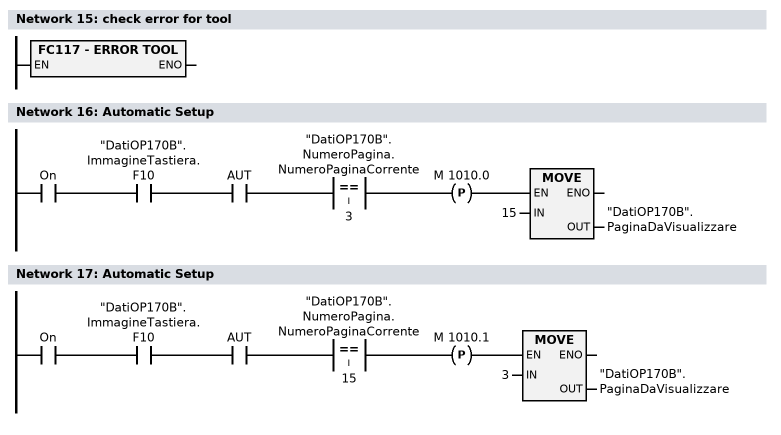
[picture p37: FC17 - OPERATOR PANNEL networks 15-17]
NETWORK
TITLE = check error for tool
      CALL  "FC117 - ERROR TOOL";
      NOP   0;
NETWORK
TITLE = Automatic Setup
      A     "On";
      A     "DatiOP170B".ImmagineTastiera.F10;
      A     "AUT";
      A(;
      L     "DatiOP170B".NumeroPagina.NumeroPaginaCorrente;
      L     3;
      ==I;
      );
      FP    M 1010.0;
      JNB   _00d;
      L     15;
      T     "DatiOP170B".PaginaDaVisualizzare;
_00d: NOP   0;
NETWORK
TITLE = Automatic Setup
      A     "On";
      A     "DatiOP170B".ImmagineTastiera.F10;
      A     "AUT";
      A(;
      L     "DatiOP170B".NumeroPagina.NumeroPaginaCorrente;
      L     15;
      ==I;
      );
      FP    M 1010.1;
      JNB   _00e;
      L     3;
      T     "DatiOP170B".PaginaDaVisualizzare;
_00e: NOP   0;
END_FUNCTION

FUNCTION "FC18 - OUTPUTS" : VOID	// FC 18
TITLE = Outputs management
VERSION : 0.1
BEGIN
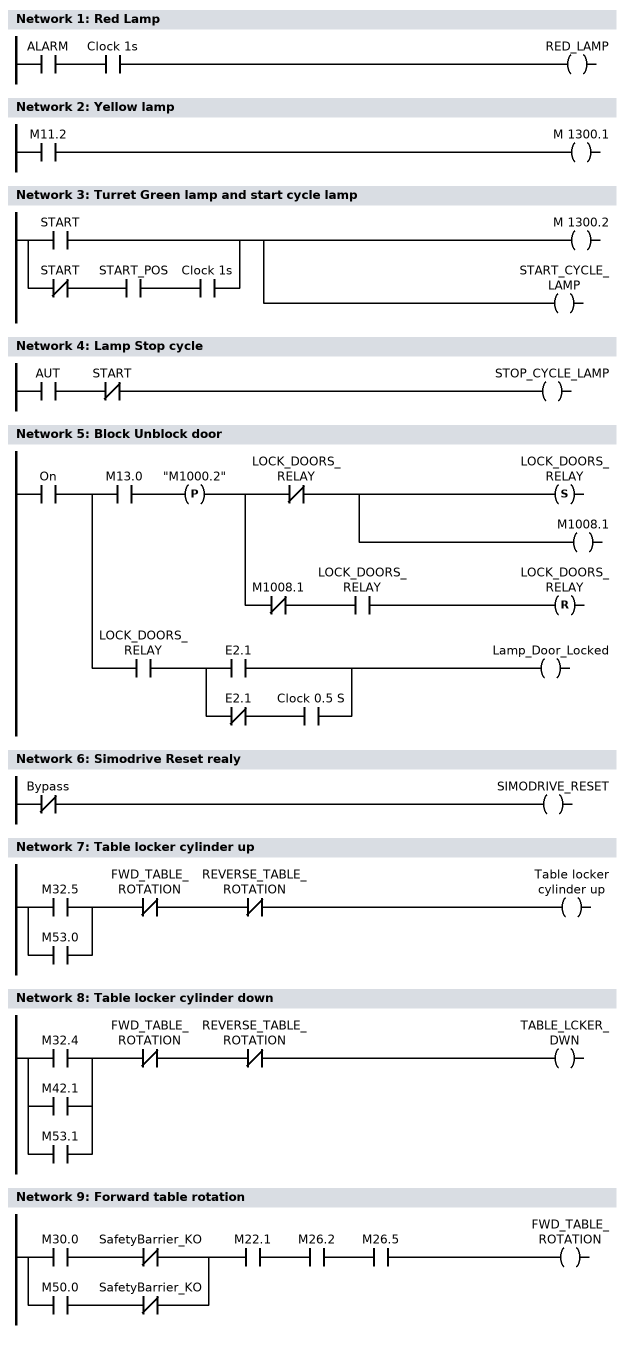
NETWORK
TITLE = Red Lamp
      A     "ALARM";
      A     "Clock 1s";
      =     "RED_LAMP";
NETWORK
TITLE = Yellow lamp
      A     "M11.2";
      =     M 1300.1;
NETWORK
TITLE = Turret Green lamp and start cycle lamp
      O     "START";
      O;
      AN    "START";
      A     "START_POS";
      A     "Clock 1s";
      =     M 1300.2;
      =     "START_CYCLE_LAMP";
NETWORK
TITLE = Lamp Stop cycle
      A     "AUT";
      AN    "START";
      =     "STOP_CYCLE_LAMP";
NETWORK
TITLE = Block Unblock door
//light ON = door lock
      A     "On";
      =     L 0.0;
      A     L 0.0;
      A     "M13.0";
      FP    "M1000.2";
      =     L 0.1;
      A     L 0.1;
      AN    "LOCK_DOORS_RELAY";
      S     "LOCK_DOORS_RELAY";
      =     "M1008.1";
      A     L 0.1;
      AN    "M1008.1";
      A     "LOCK_DOORS_RELAY";
      R     "LOCK_DOORS_RELAY";
      A     L 0.0;
      A     "LOCK_DOORS_RELAY";
      A(;
      O     "E2.1";
      O;
      AN    "E2.1";
      A     "Clock 0.5 S";
      );
      =     "Lamp_Door_Locked";
NETWORK
TITLE = Simodrive Reset realy
      AN    "Bypass";
      =     "SIMODRIVE_RESET";
NETWORK
TITLE = Table locker cylinder up
      A(;
      O     "M32.5";
      O     "M53.0";
      );
      AN    "FWD_TABLE_ROTATION";
      AN    "REVERSE_TABLE_ROTATION";
      =     "Table locker cylinder up";
NETWORK
TITLE = Table locker cylinder down
      A(;
      O     "M32.4";
      O     "M42.1";
      O     "M53.1";
      );
      AN    "FWD_TABLE_ROTATION";
      AN    "REVERSE_TABLE_ROTATION";
      =     "TABLE_LCKER_DWN";
NETWORK
TITLE = Forward table rotation
      A(;
      A     "M30.0";
      AN    "SafetyBarrier_KO";
      O;
      A     "M50.0";
      AN    "SafetyBarrier_KO";
      );
      A     "M22.1";
      A     "M26.2";
      A     "M26.5";
      =     "FWD_TABLE_ROTATION";
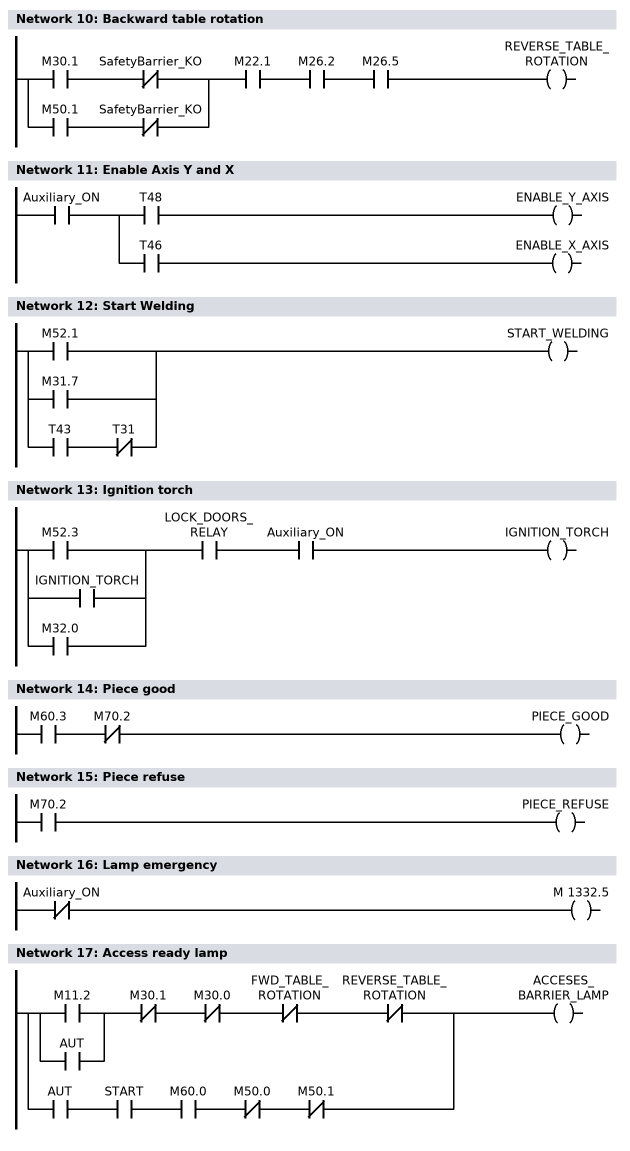
NETWORK
TITLE = Backward table rotation
      A(;
      A     "M30.1";
      AN    "SafetyBarrier_KO";
      O;
      A     "M50.1";
      AN    "SafetyBarrier_KO";
      );
      A     "M22.1";
      A     "M26.2";
      A     "M26.5";
      =     "REVERSE_TABLE_ROTATION";
NETWORK
TITLE = Enable Axis Y and X
      A     "Auxiliary_ON";
      =     L 0.0;
      A     L 0.0;
      A     "T48";
      =     "ENABLE_Y_AXIS";
      A     L 0.0;
      A     "T46";
      =     "ENABLE_X_AXIS";
NETWORK
TITLE = Start Welding
      O     "M52.1";
      O     "M31.7";
      O;
      A     "T43";
      AN    "T31";
      =     "START_WELDING";
NETWORK
TITLE = Ignition torch
      A(;
      O     "M52.3";
      O     "IGNITION_TORCH";
      O     "M32.0";
      );
      A     "LOCK_DOORS_RELAY";
      A     "Auxiliary_ON";
      =     "IGNITION_TORCH";
NETWORK
TITLE = Piece good
      A     "M60.3";
      AN    "M70.2";
      =     "PIECE_GOOD";
NETWORK
TITLE = Piece refuse
      A     "M70.2";
      =     "PIECE_REFUSE";
NETWORK
TITLE = Lamp emergency
      AN    "Auxiliary_ON";
      =     M 1332.5;
NETWORK
TITLE = Access ready lamp
      A(;
      O     "M11.2";
      O     "AUT";
      );
      AN    "M30.1";
      AN    "M30.0";
      AN    "FWD_TABLE_ROTATION";
      AN    "REVERSE_TABLE_ROTATION";
      O;
      A     "AUT";
      A     "START";
      A     "M60.0";
      AN    "M50.0";
      AN    "M50.1";
      =     "ACCESES_BARRIER_LAMP";
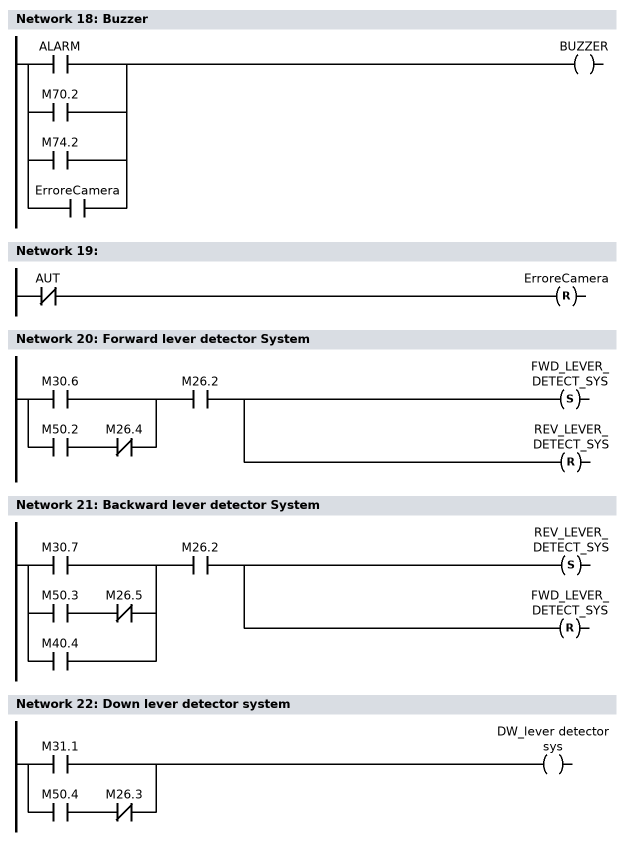
NETWORK
TITLE = Buzzer
//"Off"
      O     "ALARM";
      O     "M70.2";
      O     "M74.2";
      O     "ErroreCamera";
      =     "BUZZER";
NETWORK
TITLE =
      AN    "AUT";
      R     "ErroreCamera";
NETWORK
TITLE = Forward lever detector System
      A(;
      O     "M30.6";
      O;
      A     "M50.2";
      AN    "M26.4";
      );
      A     "M26.2";
      S     "FWD_LEVER_DETECT_SYS";
      R     "REV_LEVER_DETECT_SYS";
NETWORK
TITLE = Backward lever detector System
      A(;
      O     "M30.7";
      O;
      A     "M50.3";
      AN    "M26.5";
      O     "M40.4";
      );
      A     "M26.2";
      S     "REV_LEVER_DETECT_SYS";
      R     "FWD_LEVER_DETECT_SYS";
NETWORK
TITLE = Down lever detector system
      O     "M31.1";
      O;
      A     "M50.4";
      AN    "M26.3";
      =     "DW_lever detector sys";
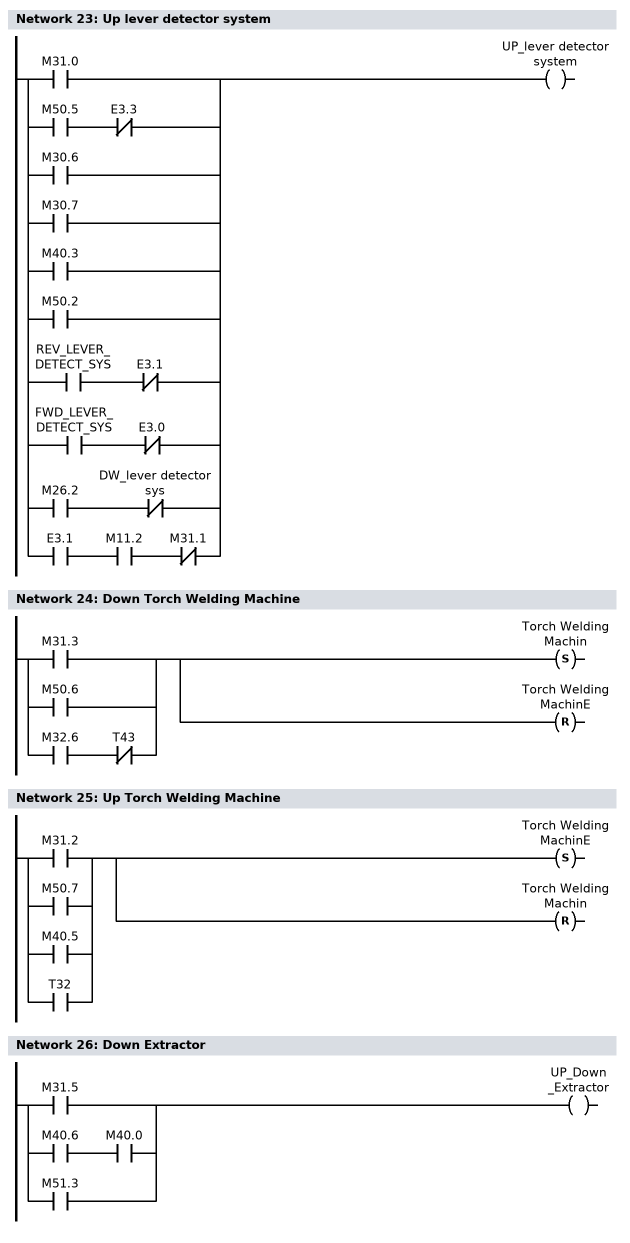
NETWORK
TITLE = Up lever detector system
      O     "M31.0";
      O;
      A     "M50.5";
      AN    "E3.3";
      O     "M30.6";
      O     "M30.7";
      O     "M40.3";
      O     "M50.2";
      O;
      A     "REV_LEVER_DETECT_SYS";
      AN    "E3.1";
      O;
      A     "FWD_LEVER_DETECT_SYS";
      AN    "E3.0";
      O;
      A     "M26.2";
      AN    "DW_lever detector sys";
      O;
      A     "E3.1";
      A     "M11.2";
      AN    "M31.1";
      =     "UP_lever detector system";
NETWORK
TITLE = Down Torch Welding Machine
      O     "M31.3";
      O     "M50.6";
      O;
      A     "M32.6";
      AN    "T43";
      S     "Torch Welding Machin";
      R     "Torch Welding MachinE";
NETWORK
TITLE = Up Torch Welding Machine
      O     "M31.2";
      O     "M50.7";
      O     "M40.5";
      O     "T32";
      S     "Torch Welding MachinE";
      R     "Torch Welding Machin";
NETWORK
TITLE = Down Extractor
      O     "M31.5";
      O;
      A     "M40.6";
      A     "M40.0";
      O     "M51.3";
      =     "UP_Down _Extractor";
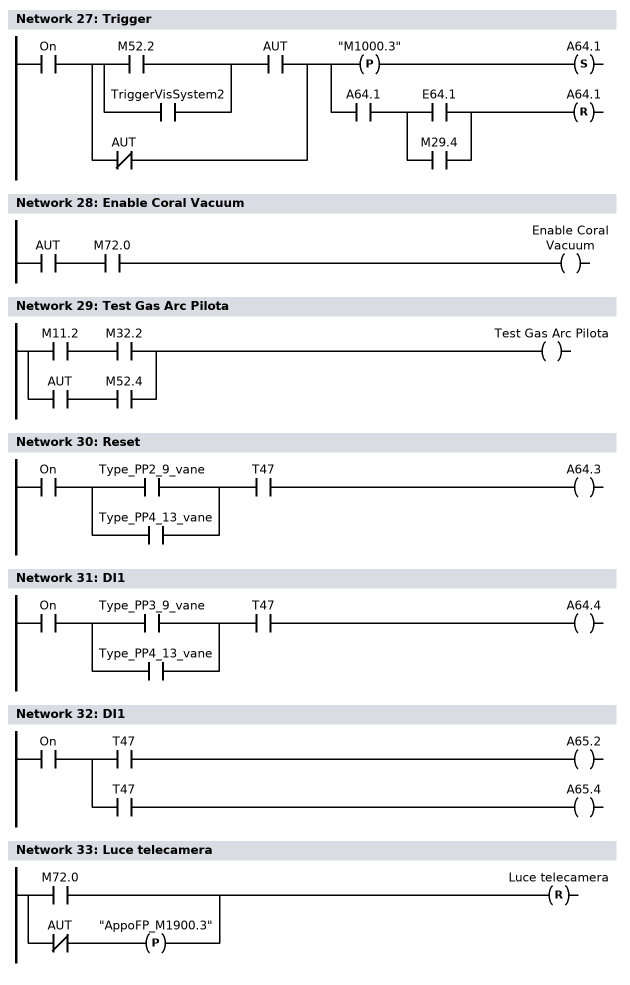
NETWORK
TITLE = Trigger
      A     "On";
      A(;
      A(;
      O     "M52.2";
      O     "TriggerVisSystem2";
      );
      A     "AUT";
      ON    "AUT";
      );
      =     L 0.0;
      A     L 0.0;
      FP    "M1000.3";
      S     "A64.1";
      A     L 0.0;
      A     "A64.1";
      A(;
      O     "E64.1";
      O     "M29.4";
      );
      R     "A64.1";
NETWORK
TITLE = Enable Coral Vacuum
      A     "AUT";
      A     "M72.0";
      =     "Enable Coral Vacuum";
NETWORK
TITLE = Test Gas Arc Pilota
//Test Arco Gas
      A     "M11.2";
      A     "M32.2";
      O;
      A     "AUT";
      A     "M52.4";
      =     "Test Gas Arc Pilota";
NETWORK
TITLE = Reset
//bit DI0 Select Scene TeleCam
      A     "On";
      A(;
      O     "Type_PP2_9_vane";
      O     "Type_PP4_13_vane";
      );
      A     "T47";
      =     "A64.3";
NETWORK
TITLE = DI1
//bit DI1 Select Scene TeleCam
      A     "On";
      A(;
      O     "Type_PP3_9_vane";
      O     "Type_PP4_13_vane";
      );
      A     "T47";
      =     "A64.4";
NETWORK
TITLE = DI1
//Select Scene Cam
      A     "On";
      =     L 0.0;
      A     L 0.0;
      A     "T47";
      =     "A65.2";
      A     L 0.0;
      A     "T47";
      =     "A65.4";
NETWORK
TITLE = Luce telecamera
      O     "M72.0";
      O(;
      AN    "AUT";
      FP    "AppoFP_M1900.3";
      );
      R     "Luce telecamera";
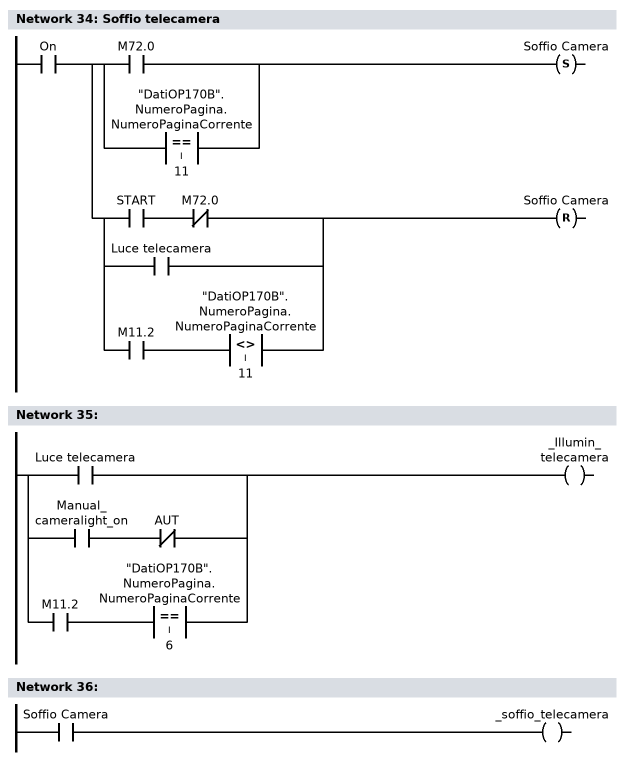
NETWORK
TITLE = Soffio telecamera
      A     "On";
      =     L 0.0;
      A     L 0.0;
      A(;
      O     "M72.0";
      O(;
      L     "DatiOP170B".NumeroPagina.NumeroPaginaCorrente;
      L     11;
      ==I;
      );
      );
      S     "Soffio Camera";
      A     L 0.0;
      A(;
      A     "START";
      AN    "M72.0";
      O     "Luce telecamera";
      O;
      A     "M11.2";
      A(;
      L     "DatiOP170B".NumeroPagina.NumeroPaginaCorrente;
      L     11;
      <>I;
      );
      );
      R     "Soffio Camera";
NETWORK
TITLE =
      O     "Luce telecamera";
      O;
      A     "Manual_cameralight_on";
      AN    "AUT";
      O;
      A     "M11.2";
      A(;
      L     "DatiOP170B".NumeroPagina.NumeroPaginaCorrente;
      L     6;
      ==I;
      );
      =     "_Illumin_telecamera";
NETWORK
TITLE =
      A     "Soffio Camera";
      =     "_soffio_telecamera";
END_FUNCTION

FUNCTION "FC19 - REPOSITIONING" : VOID	// FC 19
TITLE = Repositioning management
VERSION : 0.1
BEGIN
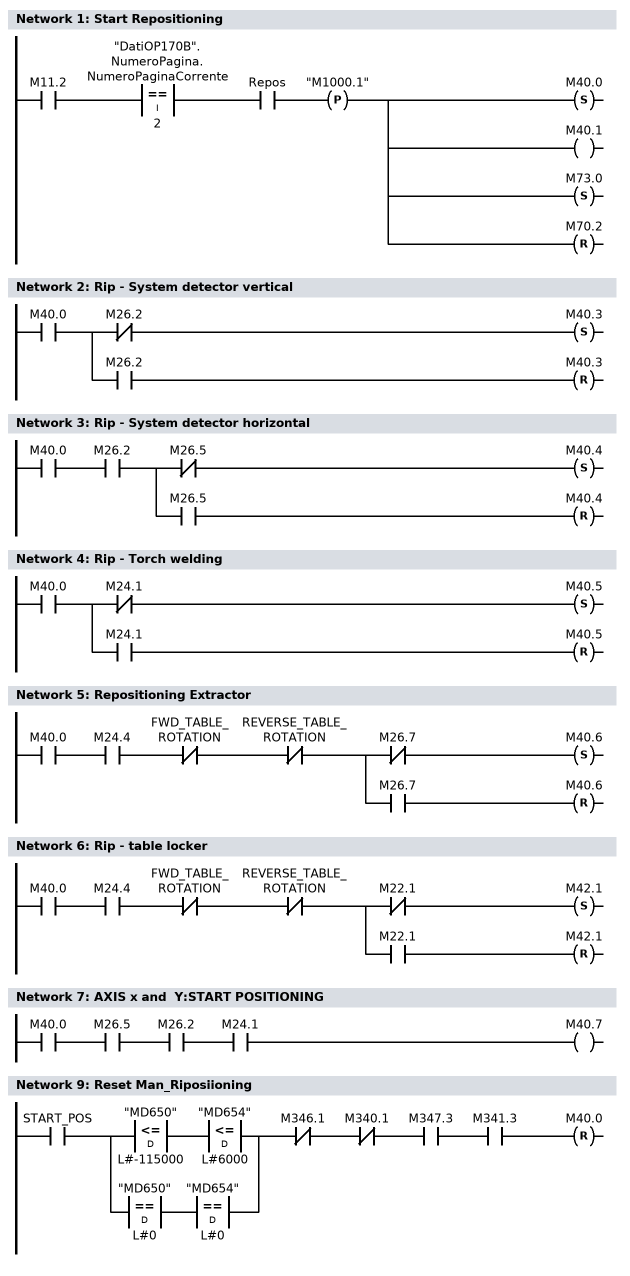
NETWORK
TITLE = Start Repositioning
      A     "M11.2";
      A(;
      L     "DatiOP170B".NumeroPagina.NumeroPaginaCorrente;
      L     2;
      ==I;
      );
      A     "Repos";
      FP    "M1000.1";
      S     "M40.0";
      =     "M40.1";
      S     "M73.0";
      R     "M70.2";
NETWORK
TITLE = Rip - System detector vertical
//ripositioning Table
      A     "M40.0";
      =     L 0.0;
      A     L 0.0;
      AN    "M26.2";
      S     "M40.3";
      A     L 0.0;
      A     "M26.2";
      R     "M40.3";
NETWORK
TITLE = Rip - System detector horizontal
//ripositioning Table
      A     "M40.0";
      A     "M26.2";
      =     L 0.0;
      A     L 0.0;
      AN    "M26.5";
      S     "M40.4";
      A     L 0.0;
      A     "M26.5";
      R     "M40.4";
NETWORK
TITLE = Rip - Torch welding
//ripositioning Table
      A     "M40.0";
      =     L 0.0;
      A     L 0.0;
      AN    "M24.1";
      S     "M40.5";
      A     L 0.0;
      A     "M24.1";
      R     "M40.5";
NETWORK
TITLE = Repositioning Extractor
      A     "M40.0";
      A     "M24.4";
      AN    "FWD_TABLE_ROTATION";
      AN    "REVERSE_TABLE_ROTATION";
      =     L 0.0;
      A     L 0.0;
      AN    "M26.7";
      S     "M40.6";
      A     L 0.0;
      A     "M26.7";
      R     "M40.6";
NETWORK
TITLE = Rip - table locker
      A     "M40.0";
      A     "M24.4";
      AN    "FWD_TABLE_ROTATION";
      AN    "REVERSE_TABLE_ROTATION";
      =     L 0.0;
      A     L 0.0;
      AN    "M22.1";
      S     "M42.1";
      A     L 0.0;
      A     "M22.1";
      R     "M42.1";
NETWORK
TITLE = AXIS x and  Y:START POSITIONING
      A     "M40.0";
      A     "M26.5";
      A     "M26.2";
      A     "M24.1";
      =     "M40.7";
NETWORK
TITLE = Reset Man_Riposiioning
//      U     "START_POS"
//      U(    
//      U(    
//      L     "MD650"
//      L     L#-115000
//      <=D   
//      )     
//      U(    
//      L     "MD654"
//      L     L#6000
//      <=D   
//      )     
//      O     
//      U(    
//      L     "MD650"
//      L     L#0
//      ==I   
//      )     
//      U(    
//      L     "MD654"
//      L     L#0
//      ==I   
//      )     
//      )     
//      UN    "M346.1"
//      UN    "M340.1"
//      U     "M347.3"
//      U     "M341.3"
//      R     "M40.0"
NETWORK
TITLE = Reset Man_Riposiioning
      A     "START_POS";
      A(;
      A(;
      L     "MD650";
      L     L#-115000;
      <=D;
      );
      A(;
      L     "MD654";
      L     L#6000;
      <=D;
      );
      O;
      A(;
      L     "MD650";
      L     L#0;
      ==D;
      );
      A(;
      L     "MD654";
      L     L#0;
      ==D;
      );
      );
      AN    "M346.1";
      AN    "M340.1";
      A     "M347.3";
      A     "M341.3";
      R     "M40.0";
NETWORK
TITLE =
END_FUNCTION

FUNCTION "FC50 - TEACH-IN" : VOID	// FC 50
TITLE = TEACH_IN
VERSION : 0.1
BEGIN
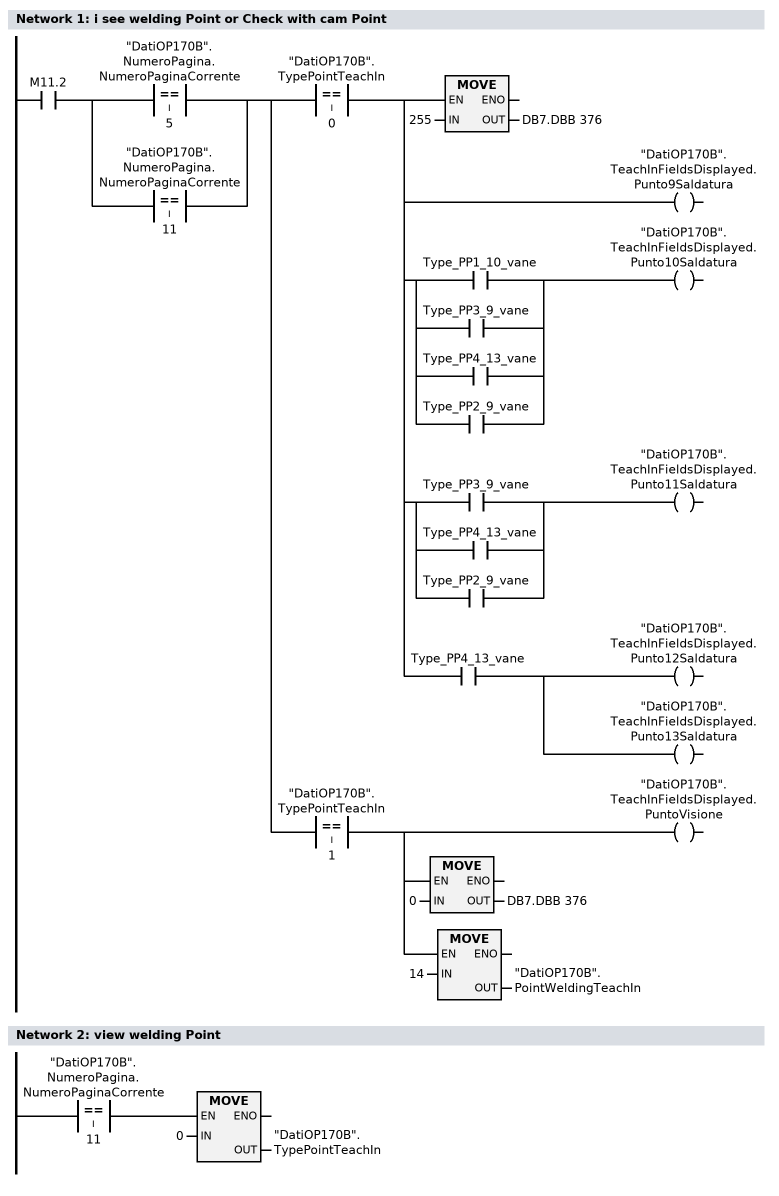
NETWORK
TITLE = i see welding Point or Check with cam Point
      A     "M11.2";
      A(;
      O(;
      L     "DatiOP170B".NumeroPagina.NumeroPaginaCorrente;
      L     5;
      ==I;
      );
      O(;
      L     "DatiOP170B".NumeroPagina.NumeroPaginaCorrente;
      L     11;
      ==I;
      );
      );
      =     L 0.0;
      A     L 0.0;
      A(;
      L     "DatiOP170B".TypePointTeachIn;
      L     0;
      ==I;
      );
      =     L 0.1;
      A     L 0.1;
      JNB   _001;
      L     255;
      T     DB7.DBB 376;
_001: NOP   0;
      A     L 0.1;
      BLD   102;
      =     "DatiOP170B".TeachInFieldsDisplayed.Punto9Saldatura;
      A     L 0.1;
      A(;
      O     "Type_PP1_10_vane";
      O     "Type_PP3_9_vane";
      O     "Type_PP4_13_vane";
      O     "Type_PP2_9_vane";
      );
      =     "DatiOP170B".TeachInFieldsDisplayed.Punto10Saldatura;
      A     L 0.1;
      A(;
      O     "Type_PP3_9_vane";
      O     "Type_PP4_13_vane";
      O     "Type_PP2_9_vane";
      );
      =     "DatiOP170B".TeachInFieldsDisplayed.Punto11Saldatura;
      A     L 0.1;
      A     "Type_PP4_13_vane";
      =     "DatiOP170B".TeachInFieldsDisplayed.Punto12Saldatura;
      =     "DatiOP170B".TeachInFieldsDisplayed.Punto13Saldatura;
      A     L 0.0;
      A(;
      L     "DatiOP170B".TypePointTeachIn;
      L     1;
      ==I;
      );
      =     L 0.1;
      A     L 0.1;
      BLD   102;
      =     "DatiOP170B".TeachInFieldsDisplayed.PuntoVisione;
      A     L 0.1;
      JNB   _002;
      L     0;
      T     DB7.DBB 376;
_002: NOP   0;
      A     L 0.1;
      JNB   _003;
      L     14;
      T     "DatiOP170B".PointWeldingTeachIn;
_003: NOP   0;
NETWORK
TITLE = view welding Point
      A(;
      L     "DatiOP170B".NumeroPagina.NumeroPaginaCorrente;
      L     11;
      ==I;
      );
      JNB   _004;
      L     0;
      T     "DatiOP170B".TypePointTeachIn;
_004: NOP   0;
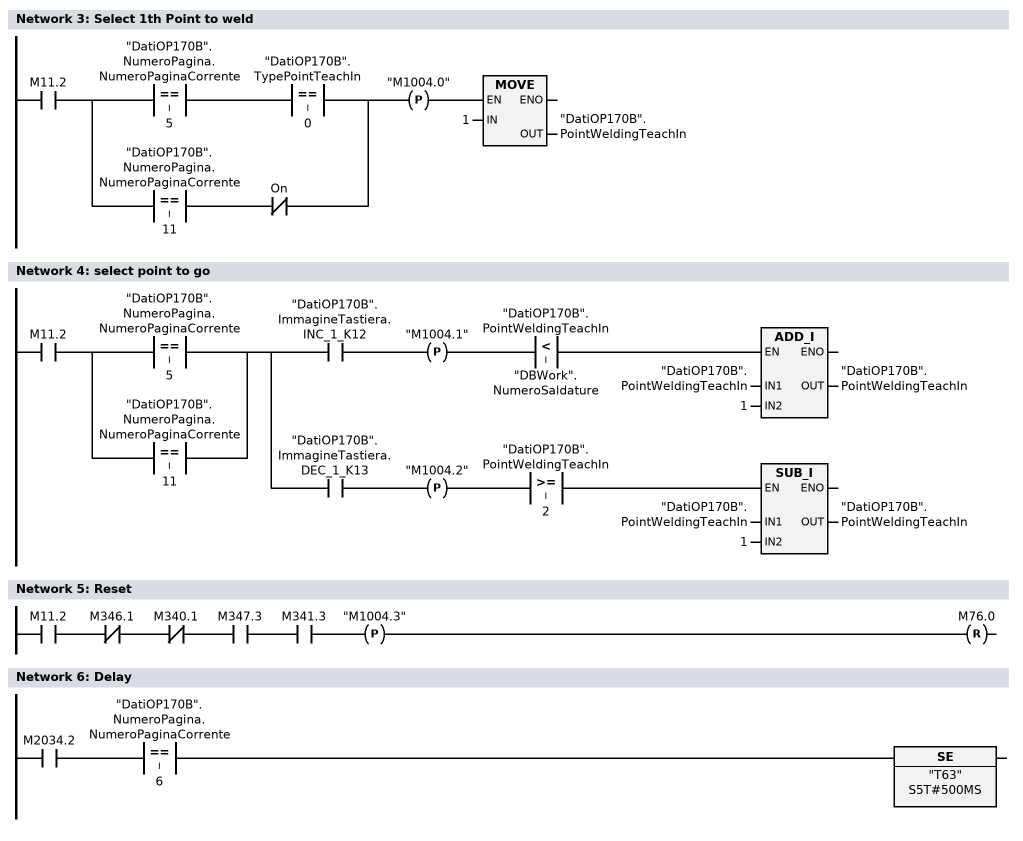
NETWORK
TITLE = Select 1th Point to weld
      A     "M11.2";
      A(;
      A(;
      L     "DatiOP170B".NumeroPagina.NumeroPaginaCorrente;
      L     5;
      ==I;
      );
      A(;
      L     "DatiOP170B".TypePointTeachIn;
      L     0;
      ==I;
      );
      O;
      A(;
      L     "DatiOP170B".NumeroPagina.NumeroPaginaCorrente;
      L     11;
      ==I;
      );
      AN    "On";
      );
      FP    "M1004.0";
      JNB   _005;
      L     1;
      T     "DatiOP170B".PointWeldingTeachIn;
_005: NOP   0;
NETWORK
TITLE = select point to go
      A     "M11.2";
      A(;
      O(;
      L     "DatiOP170B".NumeroPagina.NumeroPaginaCorrente;
      L     5;
      ==I;
      );
      O(;
      L     "DatiOP170B".NumeroPagina.NumeroPaginaCorrente;
      L     11;
      ==I;
      );
      );
      =     L 0.0;
      A     L 0.0;
      A     "DatiOP170B".ImmagineTastiera.INC_1_K12;
      FP    "M1004.1";
      A(;
      L     "DatiOP170B".PointWeldingTeachIn;
      L     "DBWork".NumeroSaldature;
      <I;
      );
      JNB   _006;
      L     "DatiOP170B".PointWeldingTeachIn;
      L     1;
      +I;
      T     "DatiOP170B".PointWeldingTeachIn;
_006: NOP   0;
      A     L 0.0;
      A     "DatiOP170B".ImmagineTastiera.DEC_1_K13;
      FP    "M1004.2";
      A(;
      L     "DatiOP170B".PointWeldingTeachIn;
      L     2;
      >=I;
      );
      JNB   _007;
      L     "DatiOP170B".PointWeldingTeachIn;
      L     1;
      -I;
      T     "DatiOP170B".PointWeldingTeachIn;
_007: NOP   0;
NETWORK
TITLE = Reset
      A     "M11.2";
      AN    "M346.1";
      AN    "M340.1";
      A     "M347.3";
      A     "M341.3";
      FP    "M1004.3";
      R     "M76.0";
NETWORK
TITLE = Delay
      A     "M2034.2";
      A(;
      L     "DatiOP170B".NumeroPagina.NumeroPaginaCorrente;
      L     6;
      ==I;
      );
      L     S5T#500MS;
      SE    "T63";
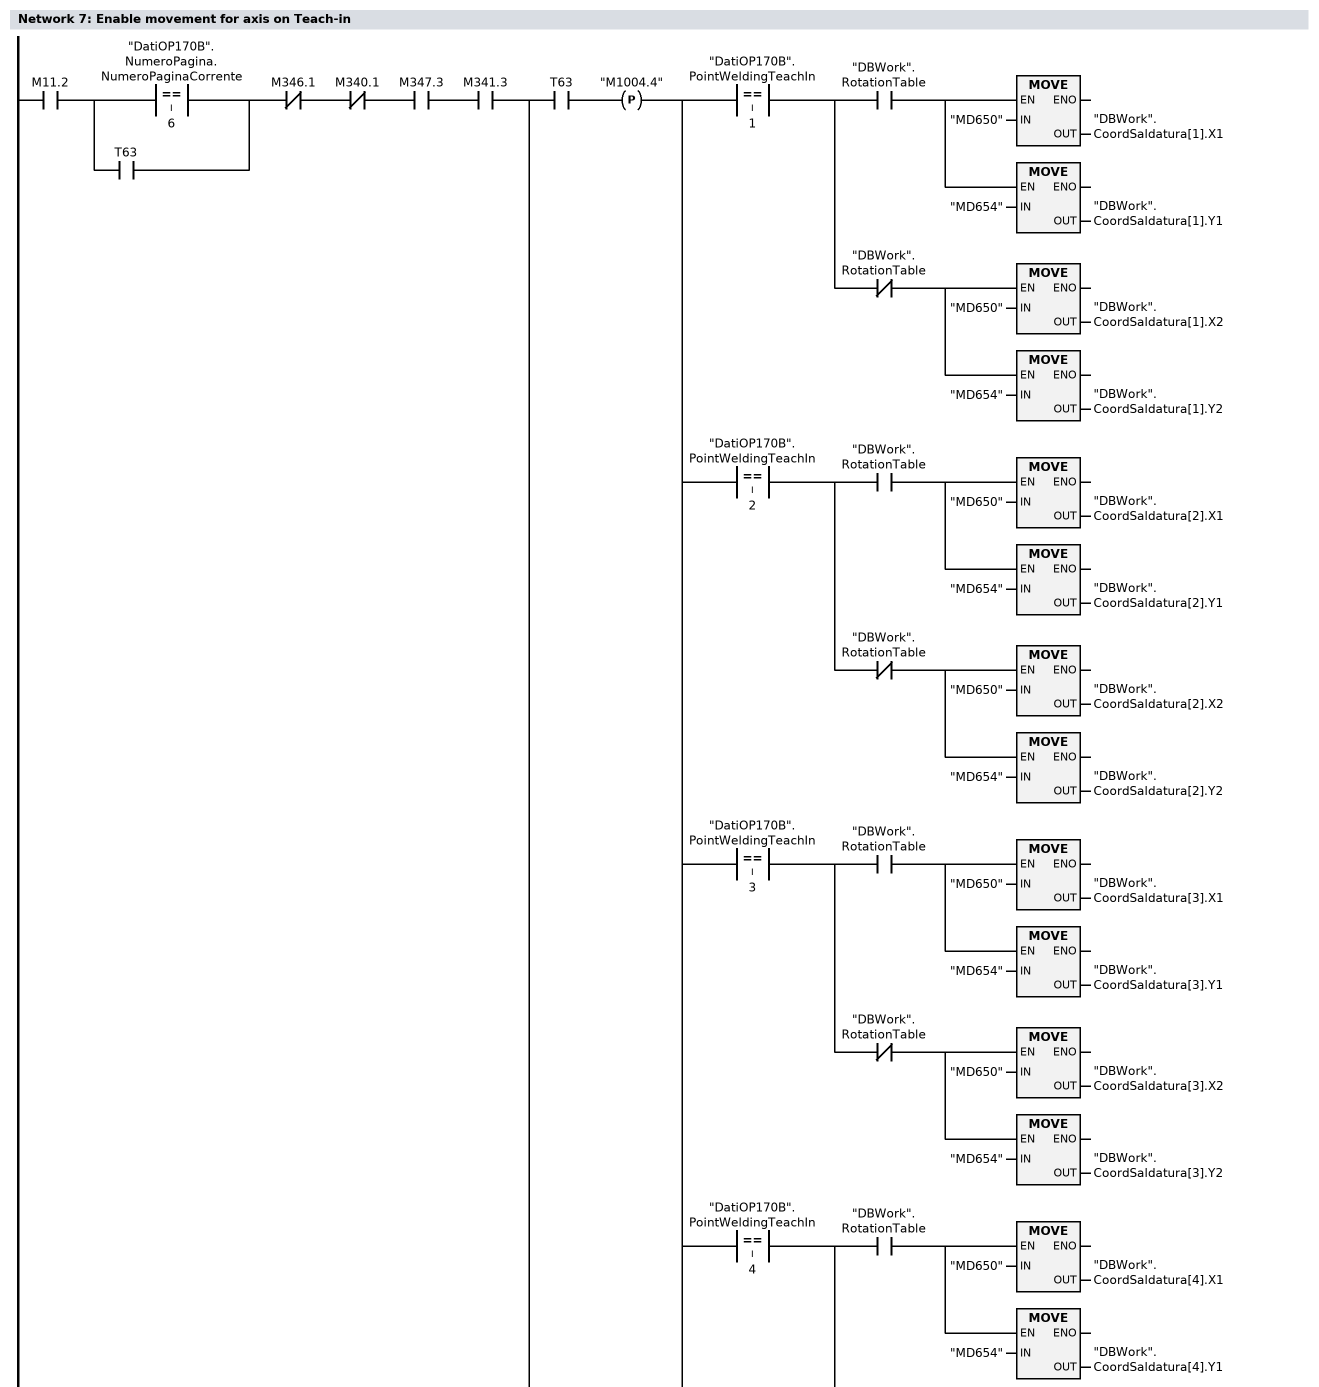
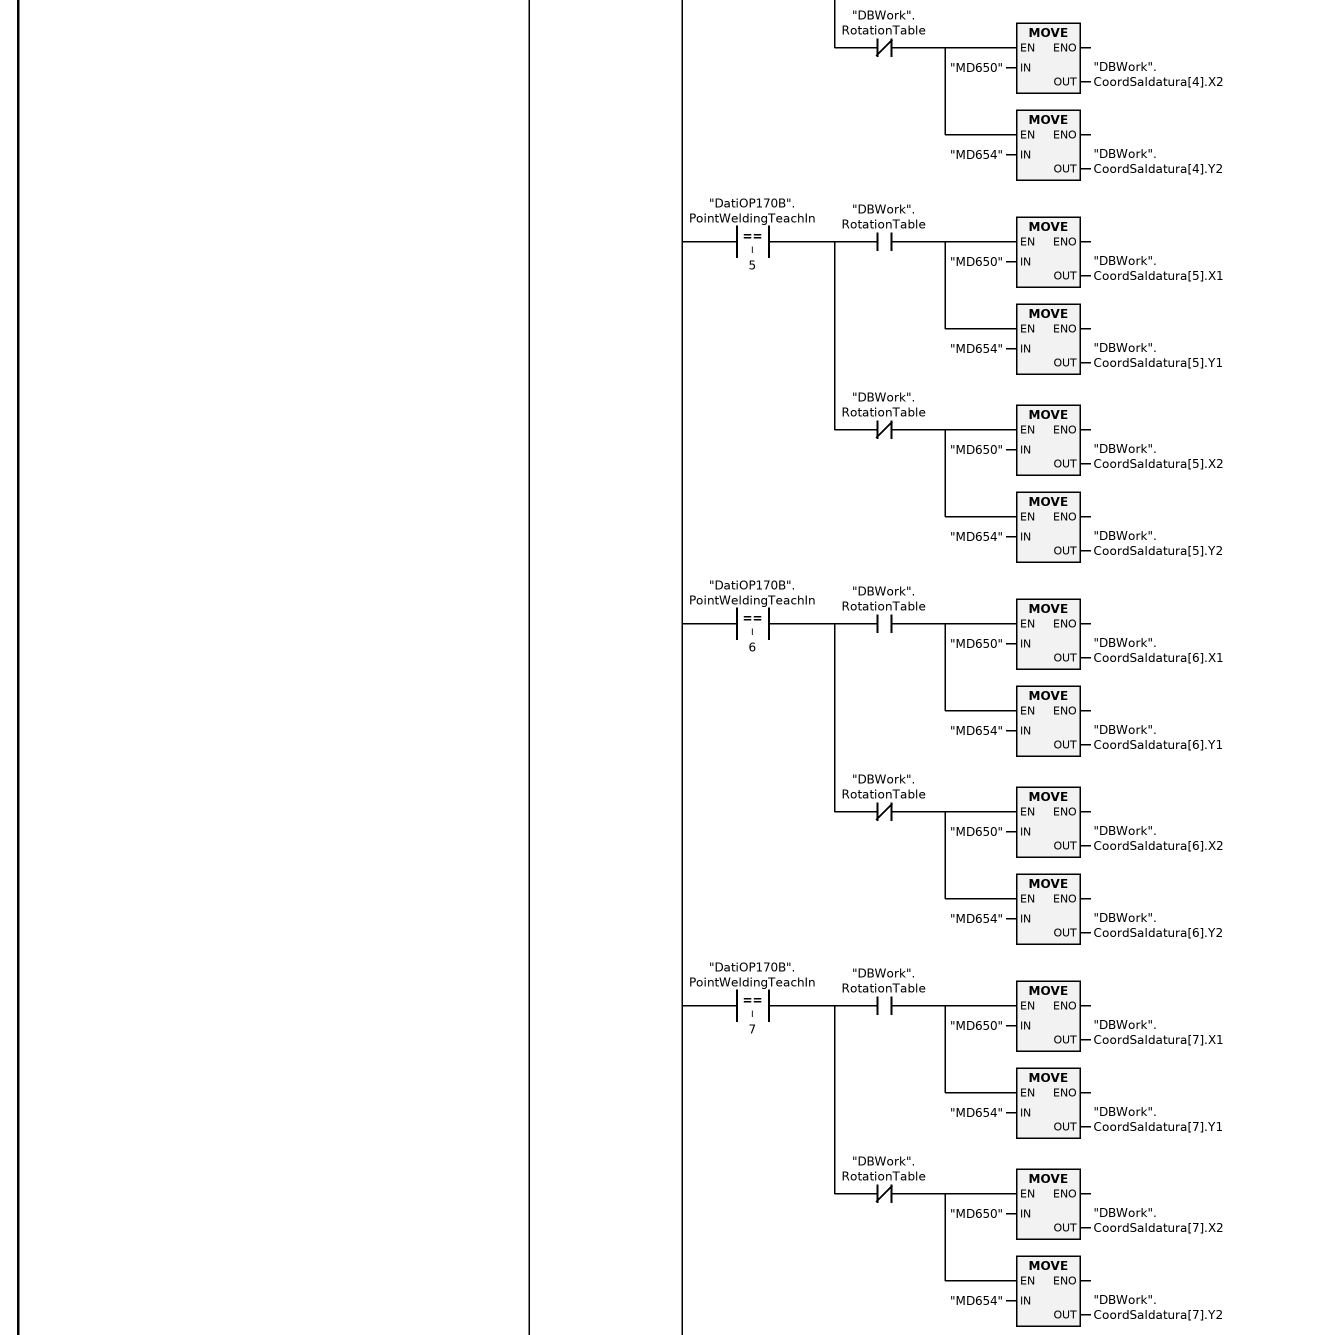
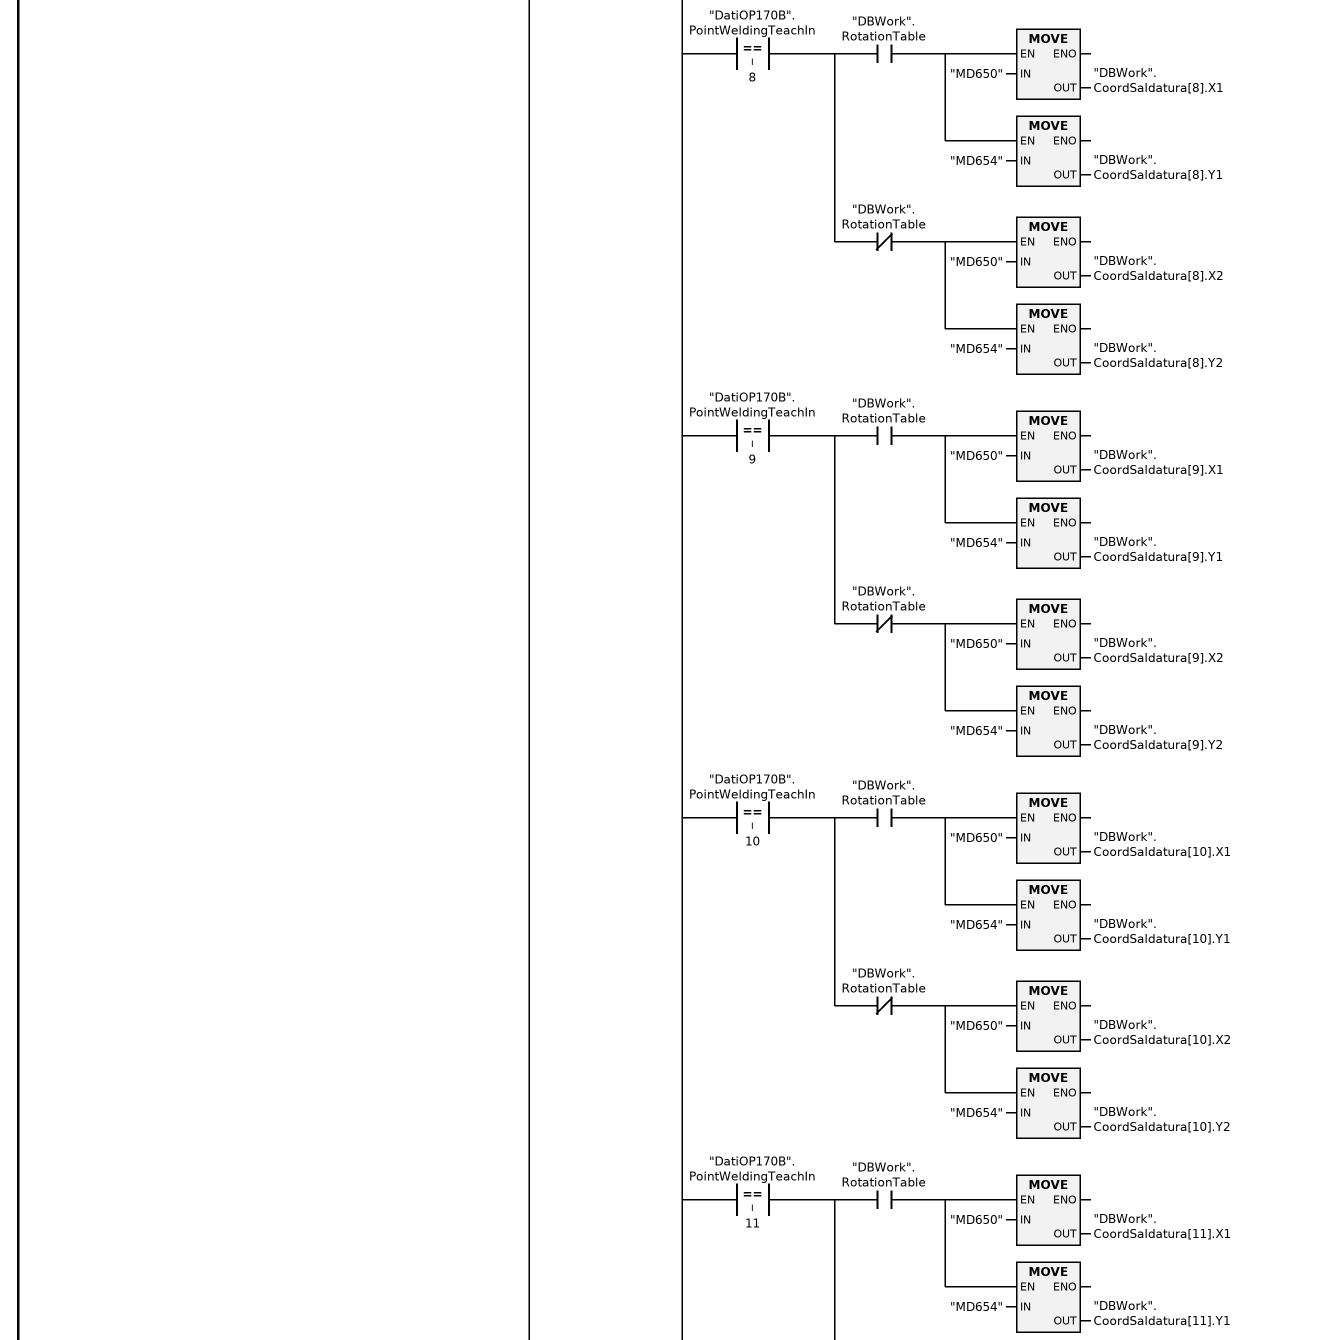
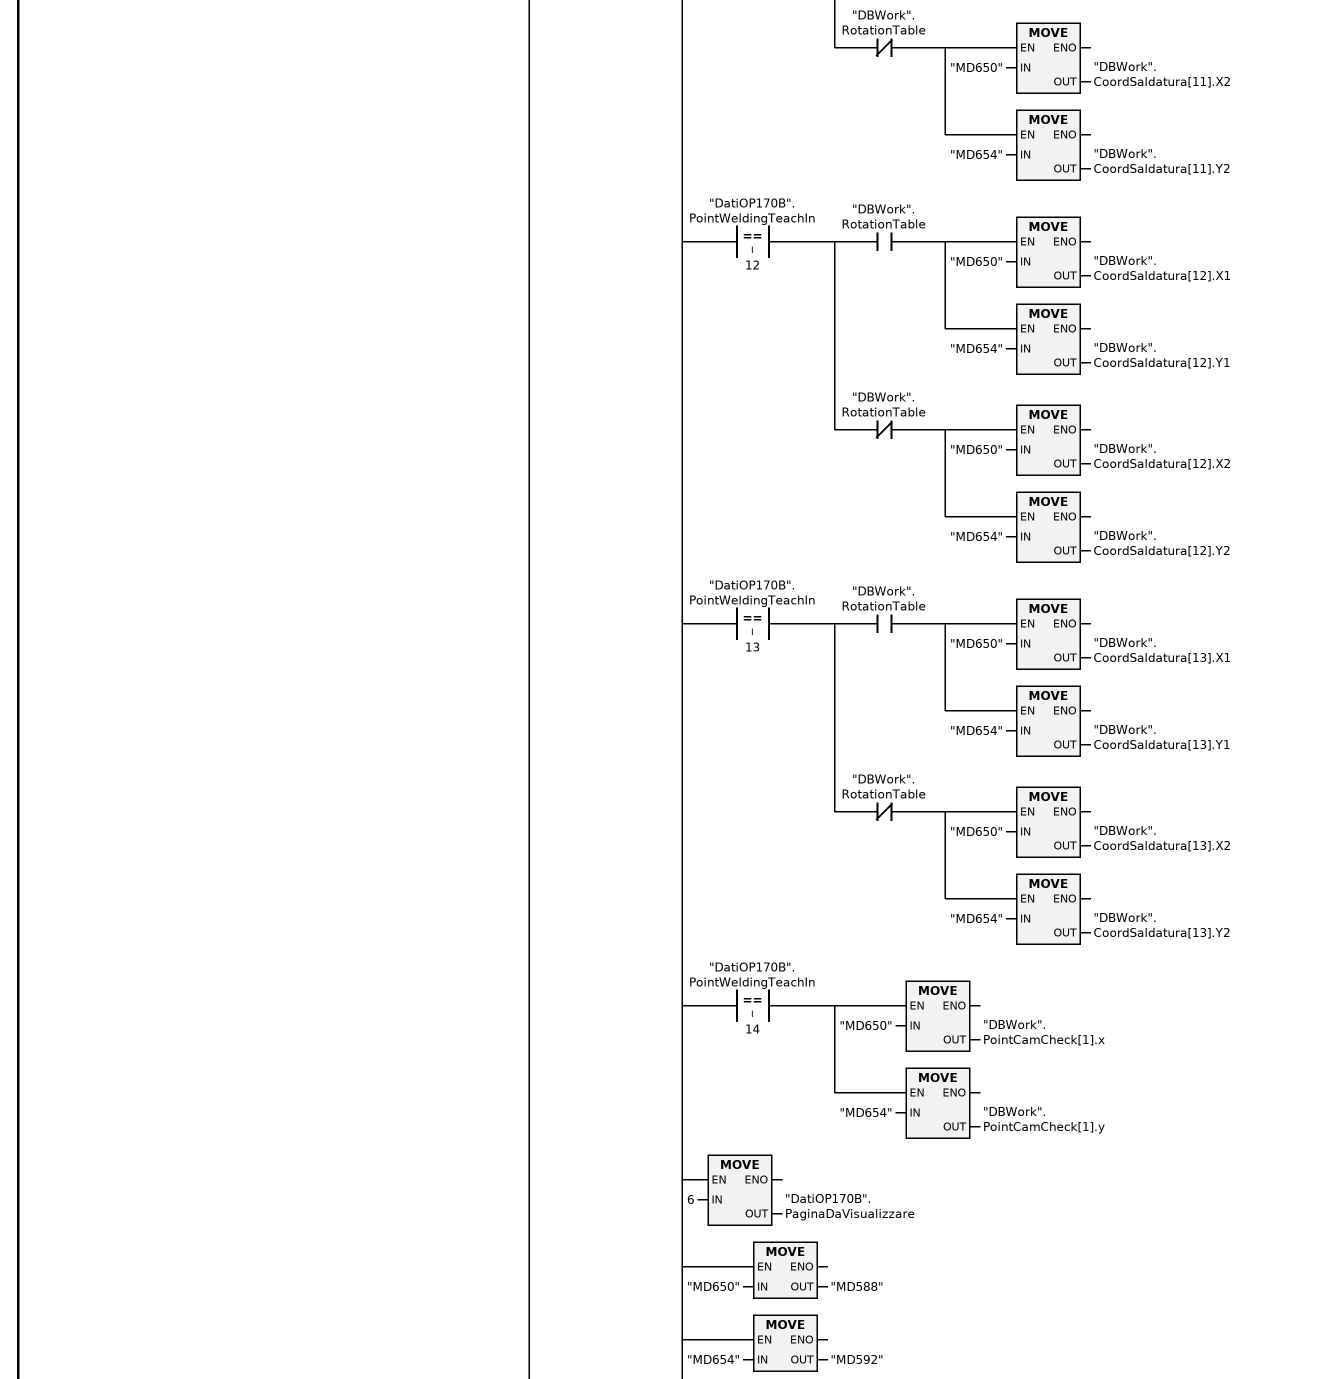
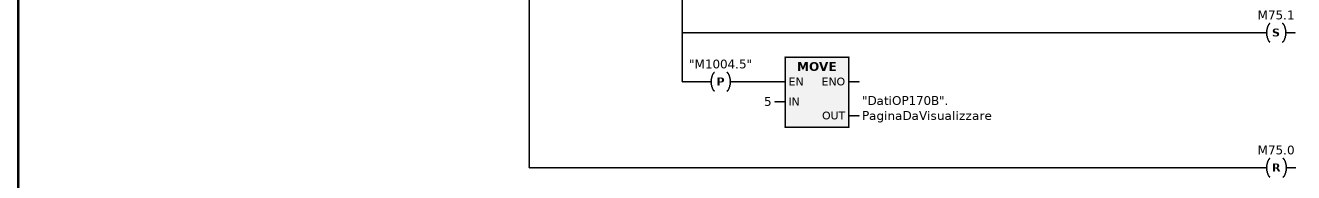
NETWORK
TITLE = Enable movement for axis on Teach-in
//move on welding point or wiev point and stored date when press teach in
//
      A     "M11.2";
      A(;
      O(;
      L     "DatiOP170B".NumeroPagina.NumeroPaginaCorrente;
      L     6;
      ==I;
      );
      O     "T63";
      );
      AN    "M346.1";
      AN    "M340.1";
      A     "M347.3";
      A     "M341.3";
      =     L 0.0;
      A     L 0.0;
      A     "T63";
      FP    "M1004.4";
      =     L 0.1;
      A     L 0.1;
      A(;
      L     "DatiOP170B".PointWeldingTeachIn;
      L     1;
      ==I;
      );
      =     L 0.2;
      A     L 0.2;
      A     "DBWork".RotationTable;
      =     L 0.3;
      A     L 0.3;
      JNB   _008;
      L     "MD650";
      T     "DBWork".CoordSaldatura[1].X1;
_008: NOP   0;
      A     L 0.3;
      JNB   _009;
      L     "MD654";
      T     "DBWork".CoordSaldatura[1].Y1;
_009: NOP   0;
      A     L 0.2;
      AN    "DBWork".RotationTable;
      =     L 0.3;
      A     L 0.3;
      JNB   _00a;
      L     "MD650";
      T     "DBWork".CoordSaldatura[1].X2;
_00a: NOP   0;
      A     L 0.3;
      JNB   _00b;
      L     "MD654";
      T     "DBWork".CoordSaldatura[1].Y2;
_00b: NOP   0;
      A     L 0.1;
      A(;
      L     "DatiOP170B".PointWeldingTeachIn;
      L     2;
      ==I;
      );
      =     L 0.2;
      A     L 0.2;
      A     "DBWork".RotationTable;
      =     L 0.3;
      A     L 0.3;
      JNB   _00c;
      L     "MD650";
      T     "DBWork".CoordSaldatura[2].X1;
_00c: NOP   0;
      A     L 0.3;
      JNB   _00d;
      L     "MD654";
      T     "DBWork".CoordSaldatura[2].Y1;
_00d: NOP   0;
      A     L 0.2;
      AN    "DBWork".RotationTable;
      =     L 0.3;
      A     L 0.3;
      JNB   _00e;
      L     "MD650";
      T     "DBWork".CoordSaldatura[2].X2;
_00e: NOP   0;
      A     L 0.3;
      JNB   _00f;
      L     "MD654";
      T     "DBWork".CoordSaldatura[2].Y2;
_00f: NOP   0;
      A     L 0.1;
      A(;
      L     "DatiOP170B".PointWeldingTeachIn;
      L     3;
      ==I;
      );
      =     L 0.2;
      A     L 0.2;
      A     "DBWork".RotationTable;
      =     L 0.3;
      A     L 0.3;
      JNB   _010;
      L     "MD650";
      T     "DBWork".CoordSaldatura[3].X1;
_010: NOP   0;
      A     L 0.3;
      JNB   _011;
      L     "MD654";
      T     "DBWork".CoordSaldatura[3].Y1;
_011: NOP   0;
      A     L 0.2;
      AN    "DBWork".RotationTable;
      =     L 0.3;
      A     L 0.3;
      JNB   _012;
      L     "MD650";
      T     "DBWork".CoordSaldatura[3].X2;
_012: NOP   0;
      A     L 0.3;
      JNB   _013;
      L     "MD654";
      T     "DBWork".CoordSaldatura[3].Y2;
_013: NOP   0;
      A     L 0.1;
      A(;
      L     "DatiOP170B".PointWeldingTeachIn;
      L     4;
      ==I;
      );
      =     L 0.2;
      A     L 0.2;
      A     "DBWork".RotationTable;
      =     L 0.3;
      A     L 0.3;
      JNB   _014;
      L     "MD650";
      T     "DBWork".CoordSaldatura[4].X1;
_014: NOP   0;
      A     L 0.3;
      JNB   _015;
      L     "MD654";
      T     "DBWork".CoordSaldatura[4].Y1;
_015: NOP   0;
      A     L 0.2;
      AN    "DBWork".RotationTable;
      =     L 0.3;
      A     L 0.3;
      JNB   _016;
      L     "MD650";
      T     "DBWork".CoordSaldatura[4].X2;
_016: NOP   0;
      A     L 0.3;
      JNB   _017;
      L     "MD654";
      T     "DBWork".CoordSaldatura[4].Y2;
_017: NOP   0;
      A     L 0.1;
      A(;
      L     "DatiOP170B".PointWeldingTeachIn;
      L     5;
      ==I;
      );
      =     L 0.2;
      A     L 0.2;
      A     "DBWork".RotationTable;
      =     L 0.3;
      A     L 0.3;
      JNB   _018;
      L     "MD650";
      T     "DBWork".CoordSaldatura[5].X1;
_018: NOP   0;
      A     L 0.3;
      JNB   _019;
      L     "MD654";
      T     "DBWork".CoordSaldatura[5].Y1;
_019: NOP   0;
      A     L 0.2;
      AN    "DBWork".RotationTable;
      =     L 0.3;
      A     L 0.3;
      JNB   _01a;
      L     "MD650";
      T     "DBWork".CoordSaldatura[5].X2;
_01a: NOP   0;
      A     L 0.3;
      JNB   _01b;
      L     "MD654";
      T     "DBWork".CoordSaldatura[5].Y2;
_01b: NOP   0;
      A     L 0.1;
      A(;
      L     "DatiOP170B".PointWeldingTeachIn;
      L     6;
      ==I;
      );
      =     L 0.2;
      A     L 0.2;
      A     "DBWork".RotationTable;
      =     L 0.3;
      A     L 0.3;
      JNB   _01c;
      L     "MD650";
      T     "DBWork".CoordSaldatura[6].X1;
_01c: NOP   0;
      A     L 0.3;
      JNB   _01d;
      L     "MD654";
      T     "DBWork".CoordSaldatura[6].Y1;
_01d: NOP   0;
      A     L 0.2;
      AN    "DBWork".RotationTable;
      =     L 0.3;
      A     L 0.3;
      JNB   _01e;
      L     "MD650";
      T     "DBWork".CoordSaldatura[6].X2;
_01e: NOP   0;
      A     L 0.3;
      JNB   _01f;
      L     "MD654";
      T     "DBWork".CoordSaldatura[6].Y2;
_01f: NOP   0;
      A     L 0.1;
      A(;
      L     "DatiOP170B".PointWeldingTeachIn;
      L     7;
      ==I;
      );
      =     L 0.2;
      A     L 0.2;
      A     "DBWork".RotationTable;
      =     L 0.3;
      A     L 0.3;
      JNB   _020;
      L     "MD650";
      T     "DBWork".CoordSaldatura[7].X1;
_020: NOP   0;
      A     L 0.3;
      JNB   _021;
      L     "MD654";
      T     "DBWork".CoordSaldatura[7].Y1;
_021: NOP   0;
      A     L 0.2;
      AN    "DBWork".RotationTable;
      =     L 0.3;
      A     L 0.3;
      JNB   _022;
      L     "MD650";
      T     "DBWork".CoordSaldatura[7].X2;
_022: NOP   0;
      A     L 0.3;
      JNB   _023;
      L     "MD654";
      T     "DBWork".CoordSaldatura[7].Y2;
_023: NOP   0;
      A     L 0.1;
      A(;
      L     "DatiOP170B".PointWeldingTeachIn;
      L     8;
      ==I;
      );
      =     L 0.2;
      A     L 0.2;
      A     "DBWork".RotationTable;
      =     L 0.3;
      A     L 0.3;
      JNB   _024;
      L     "MD650";
      T     "DBWork".CoordSaldatura[8].X1;
_024: NOP   0;
      A     L 0.3;
      JNB   _025;
      L     "MD654";
      T     "DBWork".CoordSaldatura[8].Y1;
_025: NOP   0;
      A     L 0.2;
      AN    "DBWork".RotationTable;
      =     L 0.3;
      A     L 0.3;
      JNB   _026;
      L     "MD650";
      T     "DBWork".CoordSaldatura[8].X2;
_026: NOP   0;
      A     L 0.3;
      JNB   _027;
      L     "MD654";
      T     "DBWork".CoordSaldatura[8].Y2;
_027: NOP   0;
      A     L 0.1;
      A(;
      L     "DatiOP170B".PointWeldingTeachIn;
      L     9;
      ==I;
      );
      =     L 0.2;
      A     L 0.2;
      A     "DBWork".RotationTable;
      =     L 0.3;
      A     L 0.3;
      JNB   _028;
      L     "MD650";
      T     "DBWork".CoordSaldatura[9].X1;
_028: NOP   0;
      A     L 0.3;
      JNB   _029;
      L     "MD654";
      T     "DBWork".CoordSaldatura[9].Y1;
_029: NOP   0;
      A     L 0.2;
      AN    "DBWork".RotationTable;
      =     L 0.3;
      A     L 0.3;
      JNB   _02a;
      L     "MD650";
      T     "DBWork".CoordSaldatura[9].X2;
_02a: NOP   0;
      A     L 0.3;
      JNB   _02b;
      L     "MD654";
      T     "DBWork".CoordSaldatura[9].Y2;
_02b: NOP   0;
      A     L 0.1;
      A(;
      L     "DatiOP170B".PointWeldingTeachIn;
      L     10;
      ==I;
      );
      =     L 0.2;
      A     L 0.2;
      A     "DBWork".RotationTable;
      =     L 0.3;
      A     L 0.3;
      JNB   _02c;
      L     "MD650";
      T     "DBWork".CoordSaldatura[10].X1;
_02c: NOP   0;
      A     L 0.3;
      JNB   _02d;
      L     "MD654";
      T     "DBWork".CoordSaldatura[10].Y1;
_02d: NOP   0;
      A     L 0.2;
      AN    "DBWork".RotationTable;
      =     L 0.3;
      A     L 0.3;
      JNB   _02e;
      L     "MD650";
      T     "DBWork".CoordSaldatura[10].X2;
_02e: NOP   0;
      A     L 0.3;
      JNB   _02f;
      L     "MD654";
      T     "DBWork".CoordSaldatura[10].Y2;
_02f: NOP   0;
      A     L 0.1;
      A(;
      L     "DatiOP170B".PointWeldingTeachIn;
      L     11;
      ==I;
      );
      =     L 0.2;
      A     L 0.2;
      A     "DBWork".RotationTable;
      =     L 0.3;
      A     L 0.3;
      JNB   _030;
      L     "MD650";
      T     "DBWork".CoordSaldatura[11].X1;
_030: NOP   0;
      A     L 0.3;
      JNB   _031;
      L     "MD654";
      T     "DBWork".CoordSaldatura[11].Y1;
_031: NOP   0;
      A     L 0.2;
      AN    "DBWork".RotationTable;
      =     L 0.3;
      A     L 0.3;
      JNB   _032;
      L     "MD650";
      T     "DBWork".CoordSaldatura[11].X2;
_032: NOP   0;
      A     L 0.3;
      JNB   _033;
      L     "MD654";
      T     "DBWork".CoordSaldatura[11].Y2;
_033: NOP   0;
      A     L 0.1;
      A(;
      L     "DatiOP170B".PointWeldingTeachIn;
      L     12;
      ==I;
      );
      =     L 0.2;
      A     L 0.2;
      A     "DBWork".RotationTable;
      =     L 0.3;
      A     L 0.3;
      JNB   _034;
      L     "MD650";
      T     "DBWork".CoordSaldatura[12].X1;
_034: NOP   0;
      A     L 0.3;
      JNB   _035;
      L     "MD654";
      T     "DBWork".CoordSaldatura[12].Y1;
_035: NOP   0;
      A     L 0.2;
      AN    "DBWork".RotationTable;
      =     L 0.3;
      A     L 0.3;
      JNB   _036;
      L     "MD650";
      T     "DBWork".CoordSaldatura[12].X2;
_036: NOP   0;
      A     L 0.3;
      JNB   _037;
      L     "MD654";
      T     "DBWork".CoordSaldatura[12].Y2;
_037: NOP   0;
      A     L 0.1;
      A(;
      L     "DatiOP170B".PointWeldingTeachIn;
      L     13;
      ==I;
      );
      =     L 0.2;
      A     L 0.2;
      A     "DBWork".RotationTable;
      =     L 0.3;
      A     L 0.3;
      JNB   _038;
      L     "MD650";
      T     "DBWork".CoordSaldatura[13].X1;
_038: NOP   0;
      A     L 0.3;
      JNB   _039;
      L     "MD654";
      T     "DBWork".CoordSaldatura[13].Y1;
_039: NOP   0;
      A     L 0.2;
      AN    "DBWork".RotationTable;
      =     L 0.3;
      A     L 0.3;
      JNB   _03a;
      L     "MD650";
      T     "DBWork".CoordSaldatura[13].X2;
_03a: NOP   0;
      A     L 0.3;
      JNB   _03b;
      L     "MD654";
      T     "DBWork".CoordSaldatura[13].Y2;
_03b: NOP   0;
      A     L 0.1;
      A(;
      L     "DatiOP170B".PointWeldingTeachIn;
      L     14;
      ==I;
      );
      =     L 0.2;
      A     L 0.2;
      JNB   _03c;
      L     "MD650";
      T     "DBWork".PointCamCheck[1].x;
_03c: NOP   0;
      A     L 0.2;
      JNB   _03d;
      L     "MD654";
      T     "DBWork".PointCamCheck[1].y;
_03d: NOP   0;
      A     L 0.1;
      JNB   _03e;
      L     6;
      T     "DatiOP170B".PaginaDaVisualizzare;
_03e: NOP   0;
      A     L 0.1;
      JNB   _03f;
      L     "MD650";
      T     "MD588";
_03f: NOP   0;
      A     L 0.1;
      JNB   _040;
      L     "MD654";
      T     "MD592";
_040: NOP   0;
      A     L 0.1;
      BLD   102;
      S     "M75.1";
      A     L 0.1;
      FP    "M1004.5";
      JNB   _041;
      L     5;
      T     "DatiOP170B".PaginaDaVisualizzare;
_041: NOP   0;
      A     L 0.0;
      BLD   102;
      R     "M75.0";
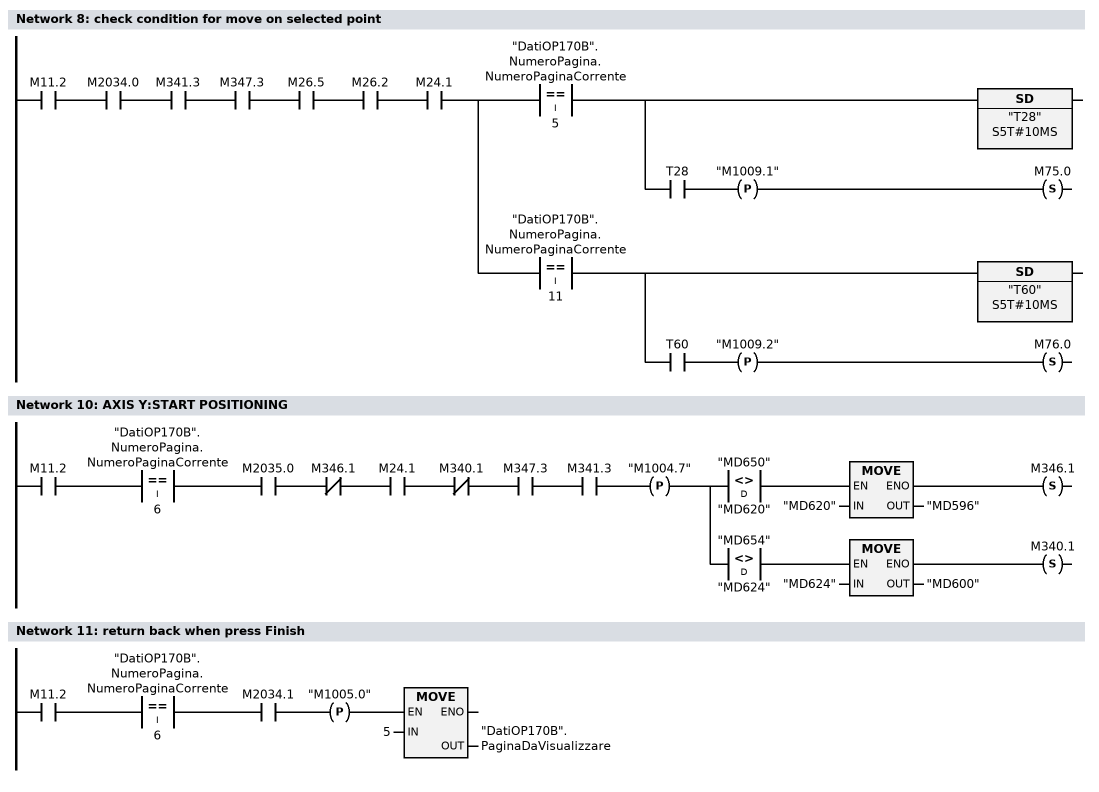
NETWORK
TITLE = check condition for move on selected point
//condition for move on selected point
      A     "M11.2";
      A     "M2034.0";
      A     "M341.3";
      A     "M347.3";
      A     "M26.5";
      A     "M26.2";
      A     "M24.1";
      =     L 0.0;
      A     L 0.0;
      A(;
      L     "DatiOP170B".NumeroPagina.NumeroPaginaCorrente;
      L     5;
      ==I;
      );
      =     L 0.1;
      A     L 0.1;
      BLD   102;
      L     S5T#10MS;
      SD    "T28";
      A     L 0.1;
      A     "T28";
      FP    "M1009.1";
      S     "M75.0";
      A     L 0.0;
      A(;
      L     "DatiOP170B".NumeroPagina.NumeroPaginaCorrente;
      L     11;
      ==I;
      );
      =     L 0.1;
      A     L 0.1;
      BLD   102;
      L     S5T#10MS;
      SD    "T60";
      A     L 0.1;
      A     "T60";
      FP    "M1009.2";
      S     "M76.0";
NETWORK
TITLE = AXIS Y:START POSITIONING
//move axis on selected point
      A     "M11.2";
      A(;
      A(;
      L     "DatiOP170B".NumeroPagina.NumeroPaginaCorrente;
      L     5;
      ==I;
      );
      A     "M75.0";
      O;
      A(;
      L     "DatiOP170B".NumeroPagina.NumeroPaginaCorrente;
      L     11;
      ==I;
      );
      A     "M76.0";
      );
      FP    "M1004.6";
      =     L 0.0;
      A     L 0.0;
      A     "DBWork".RotationTable;
      =     L 0.1;
      A(;
      A     L 0.1;
      A(;
      L     "MD588";
      L     "MD650";
      <>D;
      );
      JNB   _042;
      L     "MD588";
      L     "Timer".OffsetX1;
      +D;
      T     "MD588";
      AN    OV;
      SAVE;
      CLR;
_042: A     BR;
      );
      JNB   _043;
      L     "MD588";
      T     "MD596";
      SET;
      SAVE;
      CLR;
_043: A     BR;
      S     "M346.1";
      A(;
      A     L 0.1;
      A(;
      L     "MD592";
      L     "MD654";
      <>D;
      );
      JNB   _044;
      L     "MD592";
      L     "Timer".OffsetY1;
      +D;
      T     "MD592";
      AN    OV;
      SAVE;
      CLR;
_044: A     BR;
      );
      JNB   _045;
      L     "MD592";
      T     "MD600";
      SET;
      SAVE;
      CLR;
_045: A     BR;
      S     "M340.1";
      A     L 0.0;
      AN    "DBWork".RotationTable;
      =     L 0.1;
      A(;
      A     L 0.1;
      A(;
      L     "MD588";
      L     "MD650";
      <>D;
      );
      JNB   _046;
      L     "MD588";
      L     "DBWork2".OffsetX_2;
      +D;
      T     "MD588";
      AN    OV;
      SAVE;
      CLR;
_046: A     BR;
      );
      JNB   _047;
      L     "MD588";
      T     "MD596";
      SET;
      SAVE;
      CLR;
_047: A     BR;
      S     "M346.1";
      A(;
      A     L 0.1;
      A(;
      L     "MD592";
      L     "MD654";
      <>D;
      );
      JNB   _048;
      L     "MD592";
      L     "DBWork2".OffsetY_2;
      +D;
      T     "MD592";
      AN    OV;
      SAVE;
      CLR;
_048: A     BR;
      );
      JNB   _049;
      L     "MD592";
      T     "MD600";
      SET;
      SAVE;
      CLR;
_049: A     BR;
      S     "M340.1";
NETWORK
TITLE = AXIS Y:START POSITIONING
      A     "M11.2";
      A(;
      L     "DatiOP170B".NumeroPagina.NumeroPaginaCorrente;
      L     6;
      ==I;
      );
      A     "M2035.0";
      AN    "M346.1";
      A     "M24.1";
      AN    "M340.1";
      A     "M347.3";
      A     "M341.3";
      FP    "M1004.7";
      =     L 0.0;
      A     L 0.0;
      A(;
      L     "MD650";
      L     "MD620";
      <>D;
      );
      JNB   _04a;
      L     "MD620";
      T     "MD596";
      SET;
      SAVE;
      CLR;
_04a: A     BR;
      S     "M346.1";
      A     L 0.0;
      A(;
      L     "MD654";
      L     "MD624";
      <>D;
      );
      JNB   _04b;
      L     "MD624";
      T     "MD600";
      SET;
      SAVE;
      CLR;
_04b: A     BR;
      S     "M340.1";
NETWORK
TITLE = return back when press Finish
//retirn on previus page with finish
      A     "M11.2";
      A(;
      L     "DatiOP170B".NumeroPagina.NumeroPaginaCorrente;
      L     6;
      ==I;
      );
      A     "M2034.1";
      FP    "M1005.0";
      JNB   _04c;
      L     5;
      T     "DatiOP170B".PaginaDaVisualizzare;
_04c: NOP   0;
END_FUNCTION

FUNCTION "FC51 - TYPE TOOL" : VOID	// FC 51
VERSION : 0.1
BEGIN
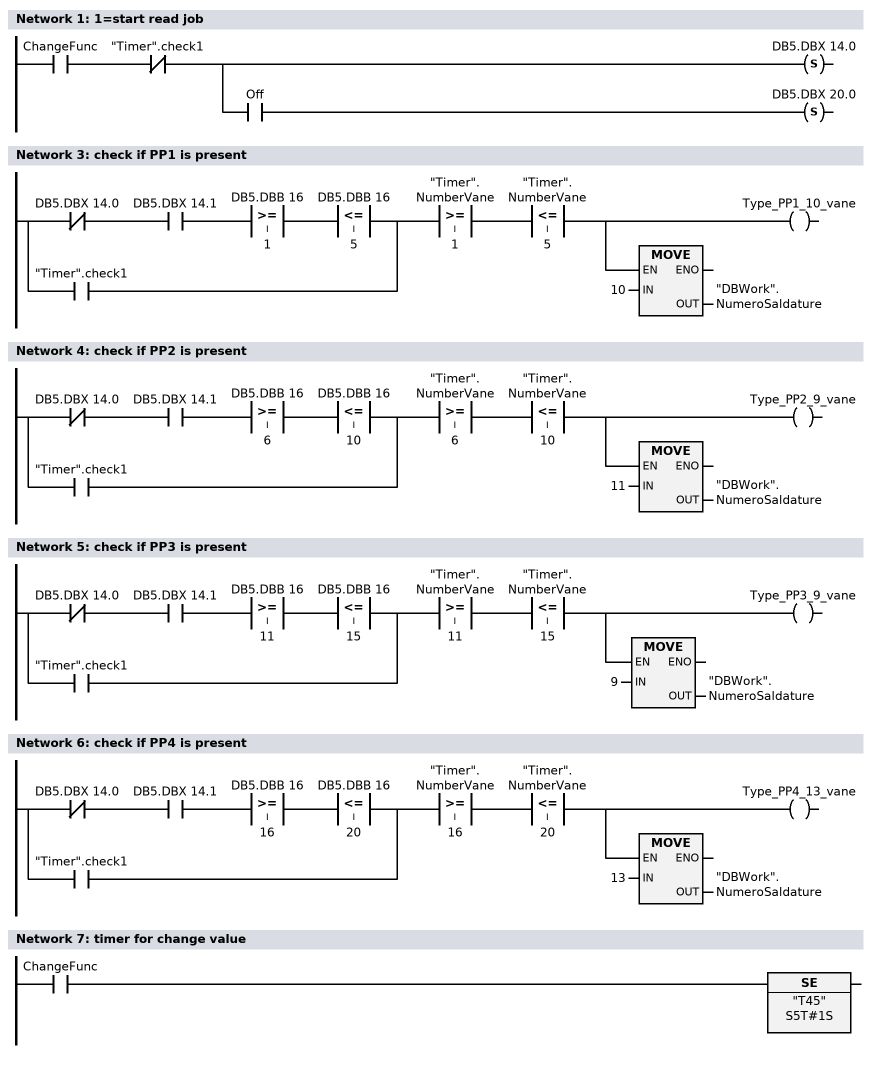
NETWORK
TITLE = 1=start read job
      A     "ChangeFunc";
      AN    "Timer".check1;
      =     L 0.0;
      A     L 0.0;
      BLD   102;
      S     DB5.DBX 14.0;
      A     L 0.0;
      A     "Off";
      S     DB5.DBX 20.0;
NETWORK
TITLE =
NETWORK
TITLE = check if PP1 is present
//Controllo se è presente il PP1
      A(;
      AN    DB5.DBX 14.0;
      A     DB5.DBX 14.1;
      A(;
      L     DB5.DBB 16;
      L     1;
      >=I;
      );
      A(;
      L     DB5.DBB 16;
      L     5;
      <=I;
      );
      O     "Timer".check1;
      );
      A(;
      L     "Timer".NumberVane;
      L     1;
      >=I;
      );
      A(;
      L     "Timer".NumberVane;
      L     5;
      <=I;
      );
      =     L 0.0;
      A     L 0.0;
      BLD   102;
      =     "Type_PP1_10_vane";
      A     L 0.0;
      JNB   _001;
      L     10;
      T     "DBWork".NumeroSaldature;
_001: NOP   0;
NETWORK
TITLE = check if PP2 is present
//Controllo se è presente il PP2
      A(;
      AN    DB5.DBX 14.0;
      A     DB5.DBX 14.1;
      A(;
      L     DB5.DBB 16;
      L     6;
      >=I;
      );
      A(;
      L     DB5.DBB 16;
      L     10;
      <=I;
      );
      O     "Timer".check1;
      );
      A(;
      L     "Timer".NumberVane;
      L     6;
      >=I;
      );
      A(;
      L     "Timer".NumberVane;
      L     10;
      <=I;
      );
      =     L 0.0;
      A     L 0.0;
      BLD   102;
      =     "Type_PP2_9_vane";
      A     L 0.0;
      JNB   _002;
      L     11;
      T     "DBWork".NumeroSaldature;
_002: NOP   0;
NETWORK
TITLE = check if PP3 is present
//Controllo se è presente il PP3
      A(;
      AN    DB5.DBX 14.0;
      A     DB5.DBX 14.1;
      A(;
      L     DB5.DBB 16;
      L     11;
      >=I;
      );
      A(;
      L     DB5.DBB 16;
      L     15;
      <=I;
      );
      O     "Timer".check1;
      );
      A(;
      L     "Timer".NumberVane;
      L     11;
      >=I;
      );
      A(;
      L     "Timer".NumberVane;
      L     15;
      <=I;
      );
      =     L 0.0;
      A     L 0.0;
      BLD   102;
      =     "Type_PP3_9_vane";
      A     L 0.0;
      JNB   _003;
      L     9;
      T     "DBWork".NumeroSaldature;
_003: NOP   0;
NETWORK
TITLE = check if PP4 is present
//Controllo se è presente il PP4
      A(;
      AN    DB5.DBX 14.0;
      A     DB5.DBX 14.1;
      A(;
      L     DB5.DBB 16;
      L     16;
      >=I;
      );
      A(;
      L     DB5.DBB 16;
      L     20;
      <=I;
      );
      O     "Timer".check1;
      );
      A(;
      L     "Timer".NumberVane;
      L     16;
      >=I;
      );
      A(;
      L     "Timer".NumberVane;
      L     20;
      <=I;
      );
      =     L 0.0;
      A     L 0.0;
      BLD   102;
      =     "Type_PP4_13_vane";
      A     L 0.0;
      JNB   _004;
      L     13;
      T     "DBWork".NumeroSaldature;
_004: NOP   0;
NETWORK
TITLE = timer for change value
      A     "ChangeFunc";
      L     S5T#1S;
      SE    "T45";
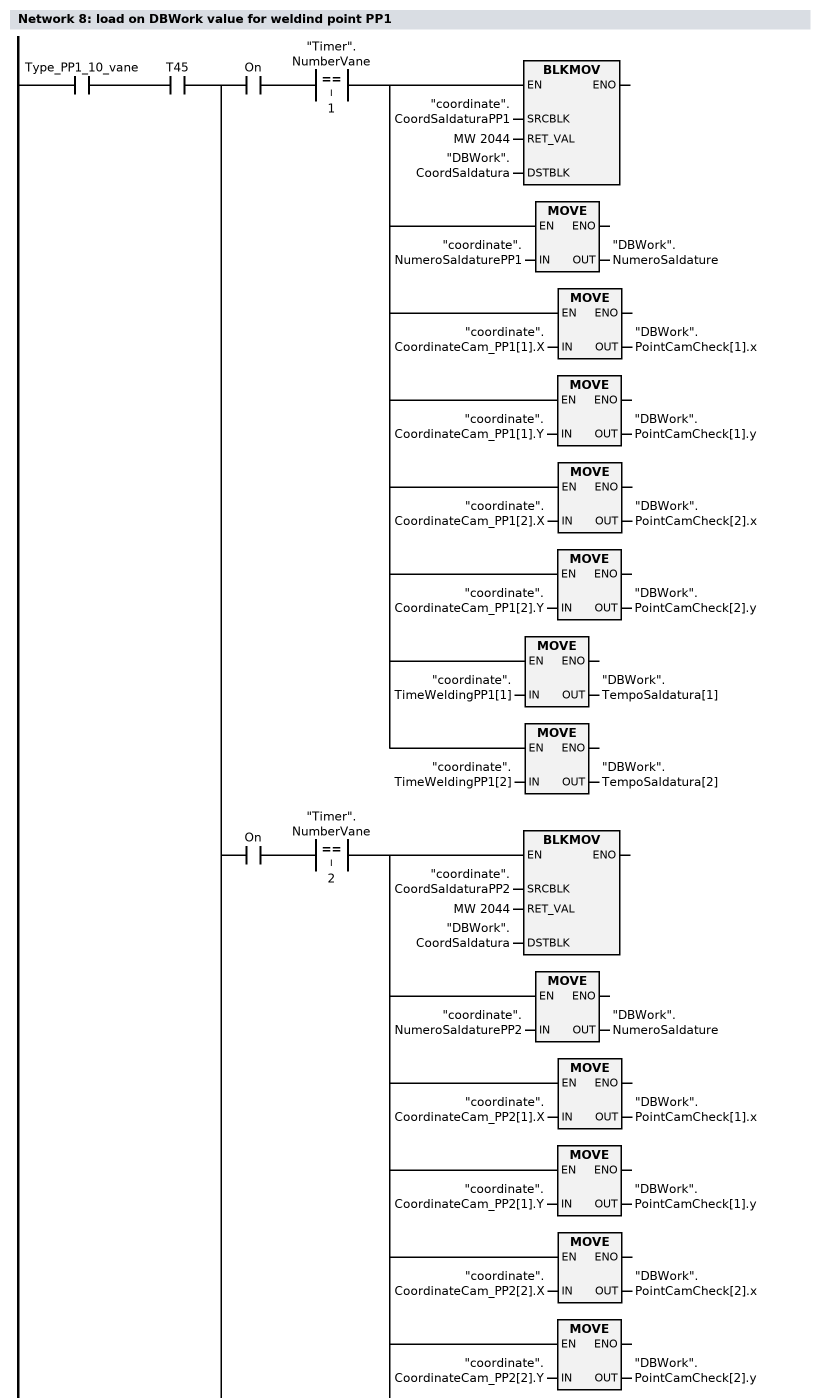
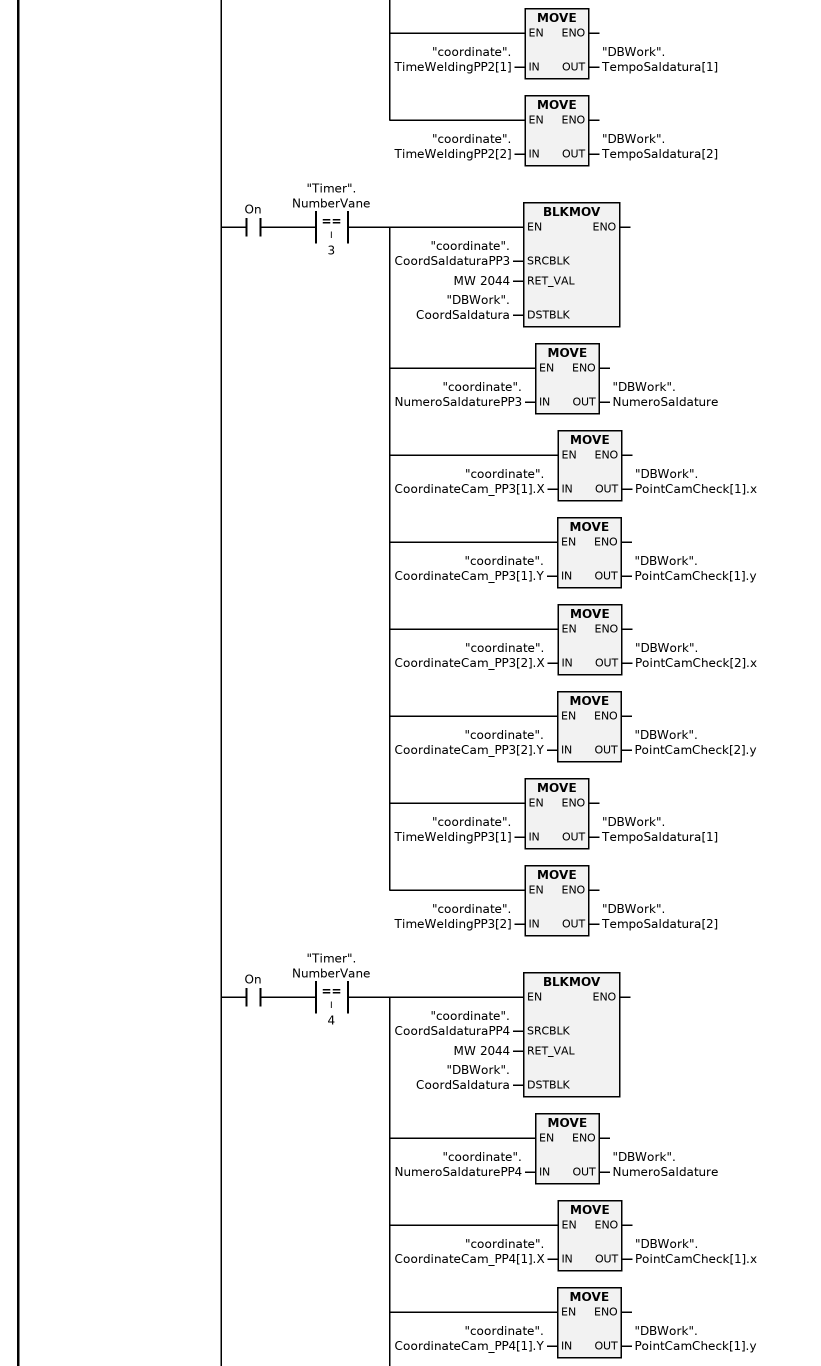
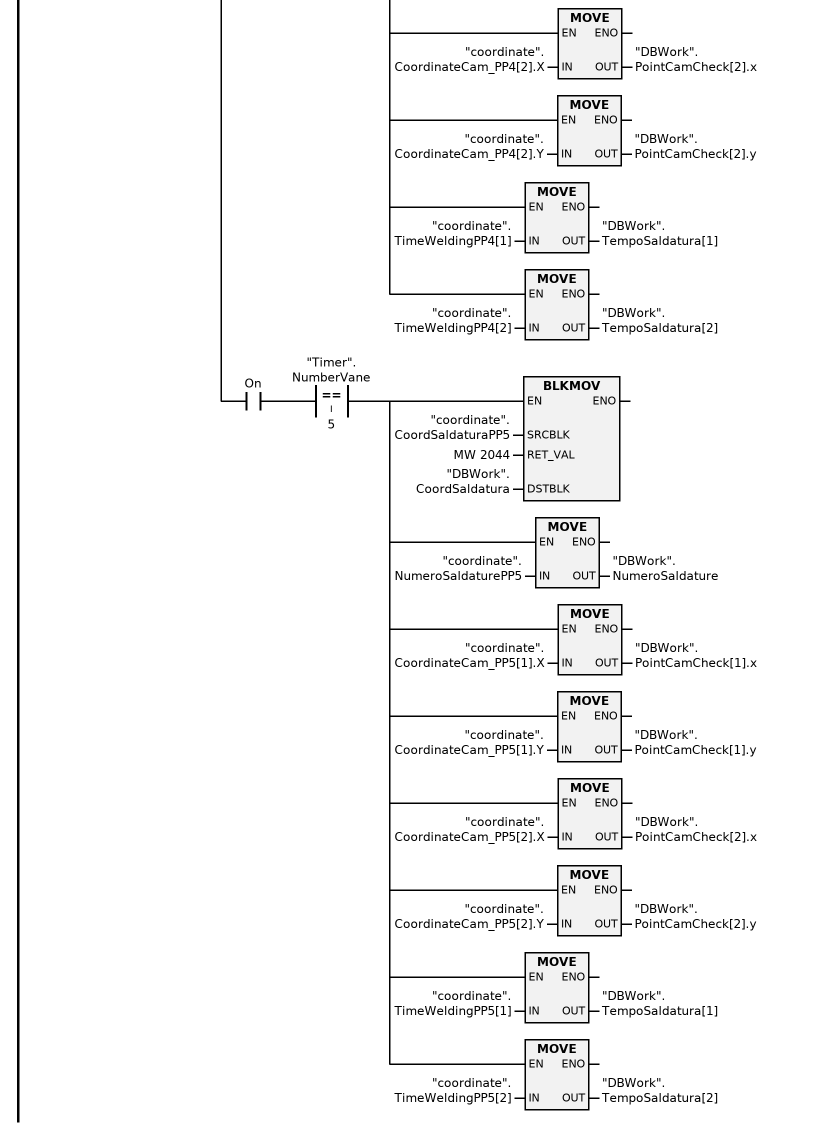
NETWORK
TITLE = load on DBWork value for weldind point PP1
//Carico sul DB Work le cordinate dei punti da saldare per il PP1
      A     "Type_PP1_10_vane";
      A     "T45";
      =     L 0.0;
      A     L 0.0;
      A     "On";
      A(;
      L     "Timer".NumberVane;
      L     1;
      ==I;
      );
      =     L 0.1;
      A     L 0.1;
      JNB   _005;
      CALL  "BLKMOV" (
           SRCBLK                   := "coordinate".CoordSaldaturaPP1,
           RET_VAL                  := MW 2044,
           DSTBLK                   := "DBWork".CoordSaldatura);
_005: NOP   0;
      A     L 0.1;
      JNB   _006;
      L     "coordinate".NumeroSaldaturePP1;
      T     "DBWork".NumeroSaldature;
_006: NOP   0;
      A     L 0.1;
      JNB   _007;
      L     "coordinate".CoordinateCam_PP1[1].X;
      T     "DBWork".PointCamCheck[1].x;
_007: NOP   0;
      A     L 0.1;
      JNB   _008;
      L     "coordinate".CoordinateCam_PP1[1].Y;
      T     "DBWork".PointCamCheck[1].y;
_008: NOP   0;
      A     L 0.1;
      JNB   _009;
      L     "coordinate".CoordinateCam_PP1[2].X;
      T     "DBWork".PointCamCheck[2].x;
_009: NOP   0;
      A     L 0.1;
      JNB   _00a;
      L     "coordinate".CoordinateCam_PP1[2].Y;
      T     "DBWork".PointCamCheck[2].y;
_00a: NOP   0;
      A     L 0.1;
      JNB   _00b;
      L     "coordinate".TimeWeldingPP1[1];
      T     "DBWork".TempoSaldatura[1];
_00b: NOP   0;
      A     L 0.1;
      JNB   _00c;
      L     "coordinate".TimeWeldingPP1[2];
      T     "DBWork".TempoSaldatura[2];
_00c: NOP   0;
      A     L 0.0;
      A     "On";
      A(;
      L     "Timer".NumberVane;
      L     2;
      ==I;
      );
      =     L 0.1;
      A     L 0.1;
      JNB   _00d;
      CALL  "BLKMOV" (
           SRCBLK                   := "coordinate".CoordSaldaturaPP2,
           RET_VAL                  := MW 2044,
           DSTBLK                   := "DBWork".CoordSaldatura);
_00d: NOP   0;
      A     L 0.1;
      JNB   _00e;
      L     "coordinate".NumeroSaldaturePP2;
      T     "DBWork".NumeroSaldature;
_00e: NOP   0;
      A     L 0.1;
      JNB   _00f;
      L     "coordinate".CoordinateCam_PP2[1].X;
      T     "DBWork".PointCamCheck[1].x;
_00f: NOP   0;
      A     L 0.1;
      JNB   _010;
      L     "coordinate".CoordinateCam_PP2[1].Y;
      T     "DBWork".PointCamCheck[1].y;
_010: NOP   0;
      A     L 0.1;
      JNB   _011;
      L     "coordinate".CoordinateCam_PP2[2].X;
      T     "DBWork".PointCamCheck[2].x;
_011: NOP   0;
      A     L 0.1;
      JNB   _012;
      L     "coordinate".CoordinateCam_PP2[2].Y;
      T     "DBWork".PointCamCheck[2].y;
_012: NOP   0;
      A     L 0.1;
      JNB   _013;
      L     "coordinate".TimeWeldingPP2[1];
      T     "DBWork".TempoSaldatura[1];
_013: NOP   0;
      A     L 0.1;
      JNB   _014;
      L     "coordinate".TimeWeldingPP2[2];
      T     "DBWork".TempoSaldatura[2];
_014: NOP   0;
      A     L 0.0;
      A     "On";
      A(;
      L     "Timer".NumberVane;
      L     3;
      ==I;
      );
      =     L 0.1;
      A     L 0.1;
      JNB   _015;
      CALL  "BLKMOV" (
           SRCBLK                   := "coordinate".CoordSaldaturaPP3,
           RET_VAL                  := MW 2044,
           DSTBLK                   := "DBWork".CoordSaldatura);
_015: NOP   0;
      A     L 0.1;
      JNB   _016;
      L     "coordinate".NumeroSaldaturePP3;
      T     "DBWork".NumeroSaldature;
_016: NOP   0;
      A     L 0.1;
      JNB   _017;
      L     "coordinate".CoordinateCam_PP3[1].X;
      T     "DBWork".PointCamCheck[1].x;
_017: NOP   0;
      A     L 0.1;
      JNB   _018;
      L     "coordinate".CoordinateCam_PP3[1].Y;
      T     "DBWork".PointCamCheck[1].y;
_018: NOP   0;
      A     L 0.1;
      JNB   _019;
      L     "coordinate".CoordinateCam_PP3[2].X;
      T     "DBWork".PointCamCheck[2].x;
_019: NOP   0;
      A     L 0.1;
      JNB   _01a;
      L     "coordinate".CoordinateCam_PP3[2].Y;
      T     "DBWork".PointCamCheck[2].y;
_01a: NOP   0;
      A     L 0.1;
      JNB   _01b;
      L     "coordinate".TimeWeldingPP3[1];
      T     "DBWork".TempoSaldatura[1];
_01b: NOP   0;
      A     L 0.1;
      JNB   _01c;
      L     "coordinate".TimeWeldingPP3[2];
      T     "DBWork".TempoSaldatura[2];
_01c: NOP   0;
      A     L 0.0;
      A     "On";
      A(;
      L     "Timer".NumberVane;
      L     4;
      ==I;
      );
      =     L 0.1;
      A     L 0.1;
      JNB   _01d;
      CALL  "BLKMOV" (
           SRCBLK                   := "coordinate".CoordSaldaturaPP4,
           RET_VAL                  := MW 2044,
           DSTBLK                   := "DBWork".CoordSaldatura);
_01d: NOP   0;
      A     L 0.1;
      JNB   _01e;
      L     "coordinate".NumeroSaldaturePP4;
      T     "DBWork".NumeroSaldature;
_01e: NOP   0;
      A     L 0.1;
      JNB   _01f;
      L     "coordinate".CoordinateCam_PP4[1].X;
      T     "DBWork".PointCamCheck[1].x;
_01f: NOP   0;
      A     L 0.1;
      JNB   _020;
      L     "coordinate".CoordinateCam_PP4[1].Y;
      T     "DBWork".PointCamCheck[1].y;
_020: NOP   0;
      A     L 0.1;
      JNB   _021;
      L     "coordinate".CoordinateCam_PP4[2].X;
      T     "DBWork".PointCamCheck[2].x;
_021: NOP   0;
      A     L 0.1;
      JNB   _022;
      L     "coordinate".CoordinateCam_PP4[2].Y;
      T     "DBWork".PointCamCheck[2].y;
_022: NOP   0;
      A     L 0.1;
      JNB   _023;
      L     "coordinate".TimeWeldingPP4[1];
      T     "DBWork".TempoSaldatura[1];
_023: NOP   0;
      A     L 0.1;
      JNB   _024;
      L     "coordinate".TimeWeldingPP4[2];
      T     "DBWork".TempoSaldatura[2];
_024: NOP   0;
      A     L 0.0;
      A     "On";
      A(;
      L     "Timer".NumberVane;
      L     5;
      ==I;
      );
      =     L 0.1;
      A     L 0.1;
      JNB   _025;
      CALL  "BLKMOV" (
           SRCBLK                   := "coordinate".CoordSaldaturaPP5,
           RET_VAL                  := MW 2044,
           DSTBLK                   := "DBWork".CoordSaldatura);
_025: NOP   0;
      A     L 0.1;
      JNB   _026;
      L     "coordinate".NumeroSaldaturePP5;
      T     "DBWork".NumeroSaldature;
_026: NOP   0;
      A     L 0.1;
      JNB   _027;
      L     "coordinate".CoordinateCam_PP5[1].X;
      T     "DBWork".PointCamCheck[1].x;
_027: NOP   0;
      A     L 0.1;
      JNB   _028;
      L     "coordinate".CoordinateCam_PP5[1].Y;
      T     "DBWork".PointCamCheck[1].y;
_028: NOP   0;
      A     L 0.1;
      JNB   _029;
      L     "coordinate".CoordinateCam_PP5[2].X;
      T     "DBWork".PointCamCheck[2].x;
_029: NOP   0;
      A     L 0.1;
      JNB   _02a;
      L     "coordinate".CoordinateCam_PP5[2].Y;
      T     "DBWork".PointCamCheck[2].y;
_02a: NOP   0;
      A     L 0.1;
      JNB   _02b;
      L     "coordinate".TimeWeldingPP5[1];
      T     "DBWork".TempoSaldatura[1];
_02b: NOP   0;
      A     L 0.1;
      JNB   _02c;
      L     "coordinate".TimeWeldingPP5[2];
      T     "DBWork".TempoSaldatura[2];
_02c: NOP   0;
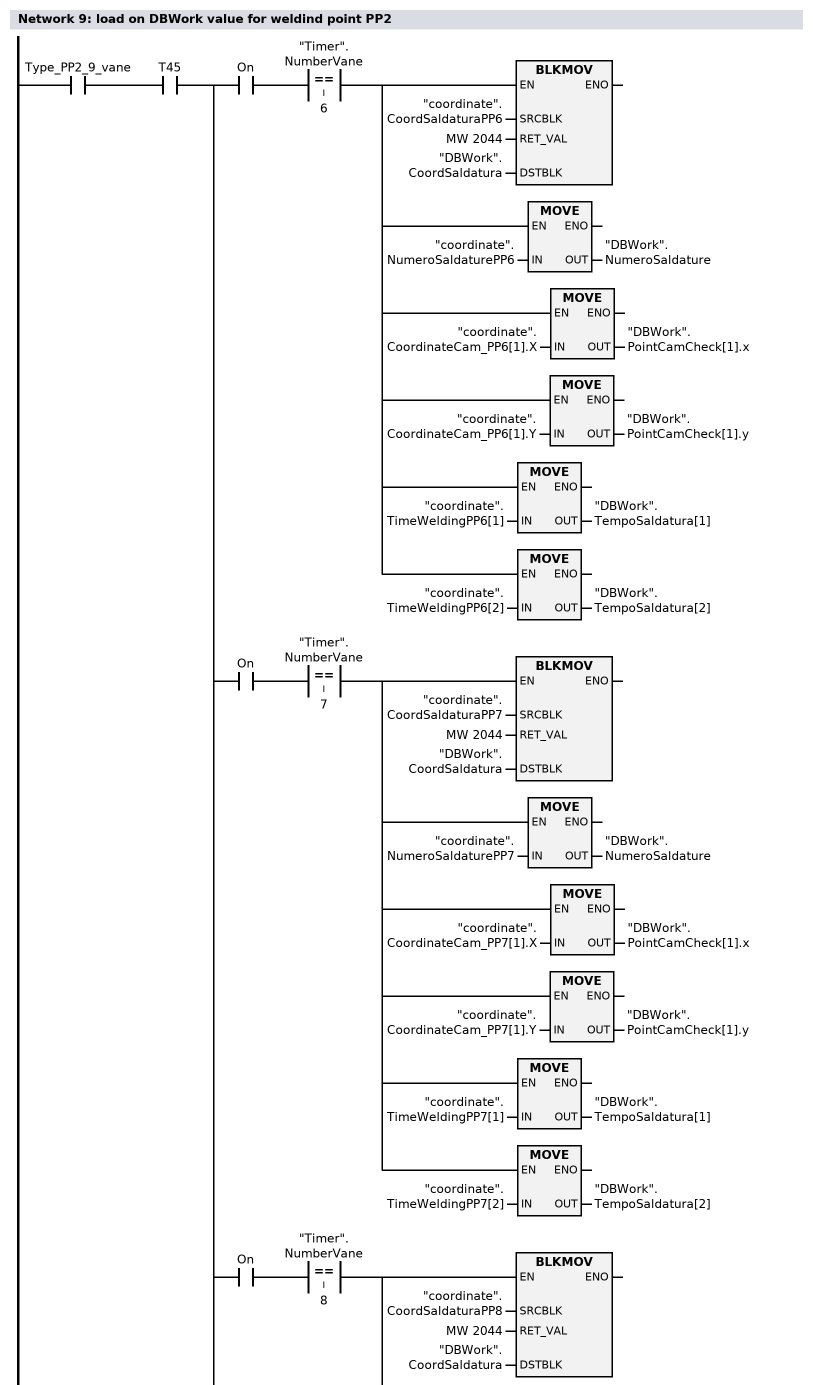
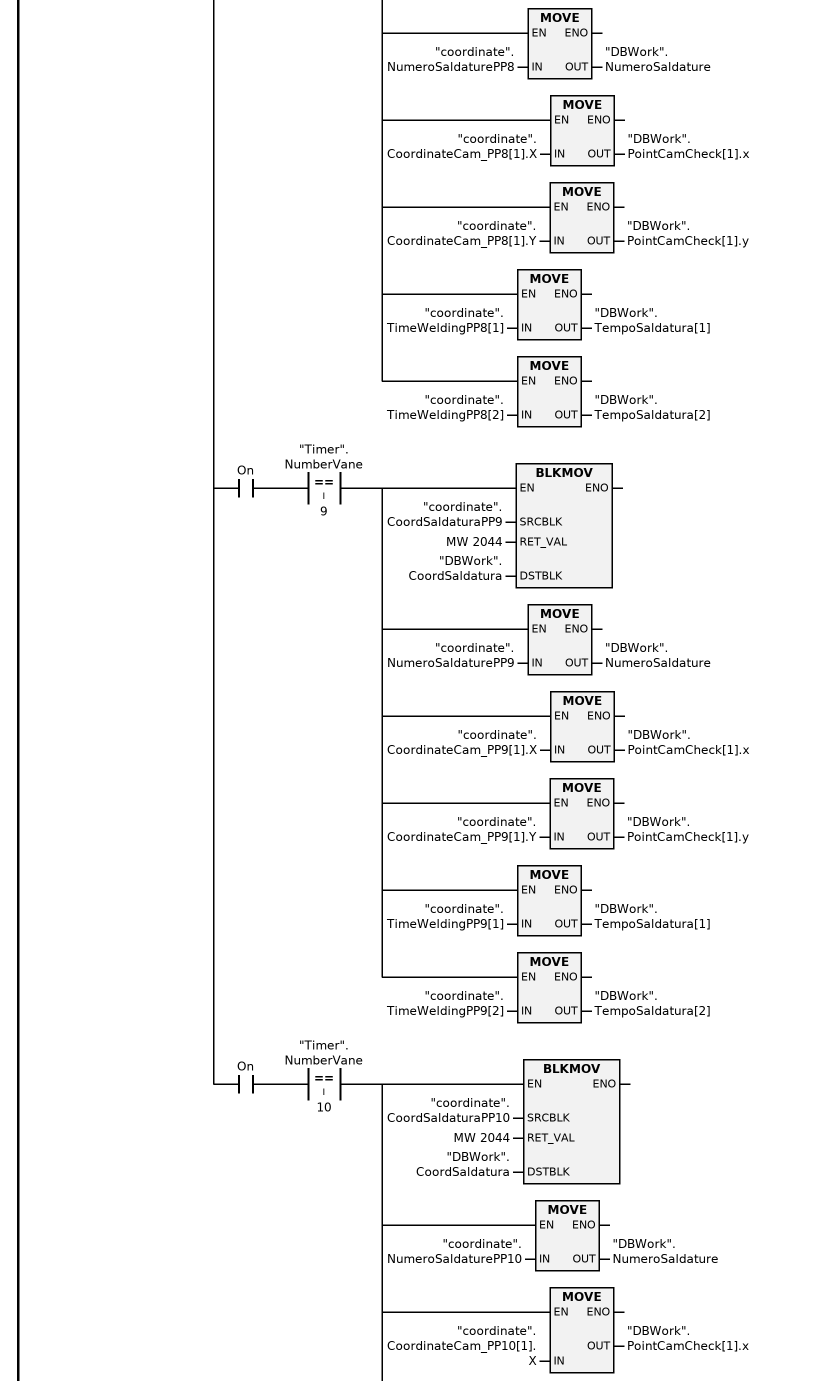
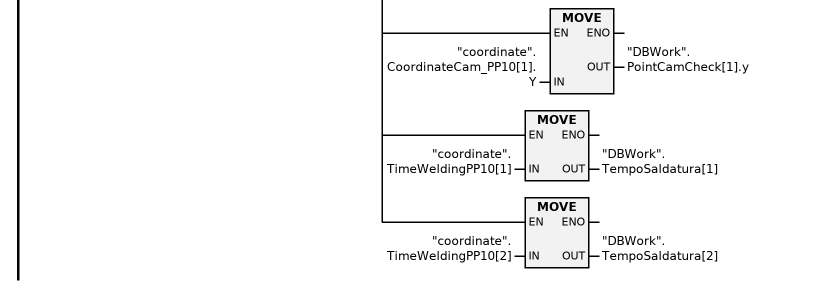
NETWORK
TITLE = load on DBWork value for weldind point PP2
//Carico sul DB Work le cordinate dei punti da saldare per il PP2
      A     "Type_PP2_9_vane";
      A     "T45";
      =     L 0.0;
      A     L 0.0;
      A     "On";
      A(;
      L     "Timer".NumberVane;
      L     6;
      ==I;
      );
      =     L 0.1;
      A     L 0.1;
      JNB   _02d;
      CALL  "BLKMOV" (
           SRCBLK                   := "coordinate".CoordSaldaturaPP6,
           RET_VAL                  := MW 2044,
           DSTBLK                   := "DBWork".CoordSaldatura);
_02d: NOP   0;
      A     L 0.1;
      JNB   _02e;
      L     "coordinate".NumeroSaldaturePP6;
      T     "DBWork".NumeroSaldature;
_02e: NOP   0;
      A     L 0.1;
      JNB   _02f;
      L     "coordinate".CoordinateCam_PP6[1].X;
      T     "DBWork".PointCamCheck[1].x;
_02f: NOP   0;
      A     L 0.1;
      JNB   _030;
      L     "coordinate".CoordinateCam_PP6[1].Y;
      T     "DBWork".PointCamCheck[1].y;
_030: NOP   0;
      A     L 0.1;
      JNB   _031;
      L     "coordinate".TimeWeldingPP6[1];
      T     "DBWork".TempoSaldatura[1];
_031: NOP   0;
      A     L 0.1;
      JNB   _032;
      L     "coordinate".TimeWeldingPP6[2];
      T     "DBWork".TempoSaldatura[2];
_032: NOP   0;
      A     L 0.0;
      A     "On";
      A(;
      L     "Timer".NumberVane;
      L     7;
      ==I;
      );
      =     L 0.1;
      A     L 0.1;
      JNB   _033;
      CALL  "BLKMOV" (
           SRCBLK                   := "coordinate".CoordSaldaturaPP7,
           RET_VAL                  := MW 2044,
           DSTBLK                   := "DBWork".CoordSaldatura);
_033: NOP   0;
      A     L 0.1;
      JNB   _034;
      L     "coordinate".NumeroSaldaturePP7;
      T     "DBWork".NumeroSaldature;
_034: NOP   0;
      A     L 0.1;
      JNB   _035;
      L     "coordinate".CoordinateCam_PP7[1].X;
      T     "DBWork".PointCamCheck[1].x;
_035: NOP   0;
      A     L 0.1;
      JNB   _036;
      L     "coordinate".CoordinateCam_PP7[1].Y;
      T     "DBWork".PointCamCheck[1].y;
_036: NOP   0;
      A     L 0.1;
      JNB   _037;
      L     "coordinate".TimeWeldingPP7[1];
      T     "DBWork".TempoSaldatura[1];
_037: NOP   0;
      A     L 0.1;
      JNB   _038;
      L     "coordinate".TimeWeldingPP7[2];
      T     "DBWork".TempoSaldatura[2];
_038: NOP   0;
      A     L 0.0;
      A     "On";
      A(;
      L     "Timer".NumberVane;
      L     8;
      ==I;
      );
      =     L 0.1;
      A     L 0.1;
      JNB   _039;
      CALL  "BLKMOV" (
           SRCBLK                   := "coordinate".CoordSaldaturaPP8,
           RET_VAL                  := MW 2044,
           DSTBLK                   := "DBWork".CoordSaldatura);
_039: NOP   0;
      A     L 0.1;
      JNB   _03a;
      L     "coordinate".NumeroSaldaturePP8;
      T     "DBWork".NumeroSaldature;
_03a: NOP   0;
      A     L 0.1;
      JNB   _03b;
      L     "coordinate".CoordinateCam_PP8[1].X;
      T     "DBWork".PointCamCheck[1].x;
_03b: NOP   0;
      A     L 0.1;
      JNB   _03c;
      L     "coordinate".CoordinateCam_PP8[1].Y;
      T     "DBWork".PointCamCheck[1].y;
_03c: NOP   0;
      A     L 0.1;
      JNB   _03d;
      L     "coordinate".TimeWeldingPP8[1];
      T     "DBWork".TempoSaldatura[1];
_03d: NOP   0;
      A     L 0.1;
      JNB   _03e;
      L     "coordinate".TimeWeldingPP8[2];
      T     "DBWork".TempoSaldatura[2];
_03e: NOP   0;
      A     L 0.0;
      A     "On";
      A(;
      L     "Timer".NumberVane;
      L     9;
      ==I;
      );
      =     L 0.1;
      A     L 0.1;
      JNB   _03f;
      CALL  "BLKMOV" (
           SRCBLK                   := "coordinate".CoordSaldaturaPP9,
           RET_VAL                  := MW 2044,
           DSTBLK                   := "DBWork".CoordSaldatura);
_03f: NOP   0;
      A     L 0.1;
      JNB   _040;
      L     "coordinate".NumeroSaldaturePP9;
      T     "DBWork".NumeroSaldature;
_040: NOP   0;
      A     L 0.1;
      JNB   _041;
      L     "coordinate".CoordinateCam_PP9[1].X;
      T     "DBWork".PointCamCheck[1].x;
_041: NOP   0;
      A     L 0.1;
      JNB   _042;
      L     "coordinate".CoordinateCam_PP9[1].Y;
      T     "DBWork".PointCamCheck[1].y;
_042: NOP   0;
      A     L 0.1;
      JNB   _043;
      L     "coordinate".TimeWeldingPP9[1];
      T     "DBWork".TempoSaldatura[1];
_043: NOP   0;
      A     L 0.1;
      JNB   _044;
      L     "coordinate".TimeWeldingPP9[2];
      T     "DBWork".TempoSaldatura[2];
_044: NOP   0;
      A     L 0.0;
      A     "On";
      A(;
      L     "Timer".NumberVane;
      L     10;
      ==I;
      );
      =     L 0.1;
      A     L 0.1;
      JNB   _045;
      CALL  "BLKMOV" (
           SRCBLK                   := "coordinate".CoordSaldaturaPP10,
           RET_VAL                  := MW 2044,
           DSTBLK                   := "DBWork".CoordSaldatura);
_045: NOP   0;
      A     L 0.1;
      JNB   _046;
      L     "coordinate".NumeroSaldaturePP10;
      T     "DBWork".NumeroSaldature;
_046: NOP   0;
      A     L 0.1;
      JNB   _047;
      L     "coordinate".CoordinateCam_PP10[1].X;
      T     "DBWork".PointCamCheck[1].x;
_047: NOP   0;
      A     L 0.1;
      JNB   _048;
      L     "coordinate".CoordinateCam_PP10[1].Y;
      T     "DBWork".PointCamCheck[1].y;
_048: NOP   0;
      A     L 0.1;
      JNB   _049;
      L     "coordinate".TimeWeldingPP10[1];
      T     "DBWork".TempoSaldatura[1];
_049: NOP   0;
      A     L 0.1;
      JNB   _04a;
      L     "coordinate".TimeWeldingPP10[2];
      T     "DBWork".TempoSaldatura[2];
_04a: NOP   0;
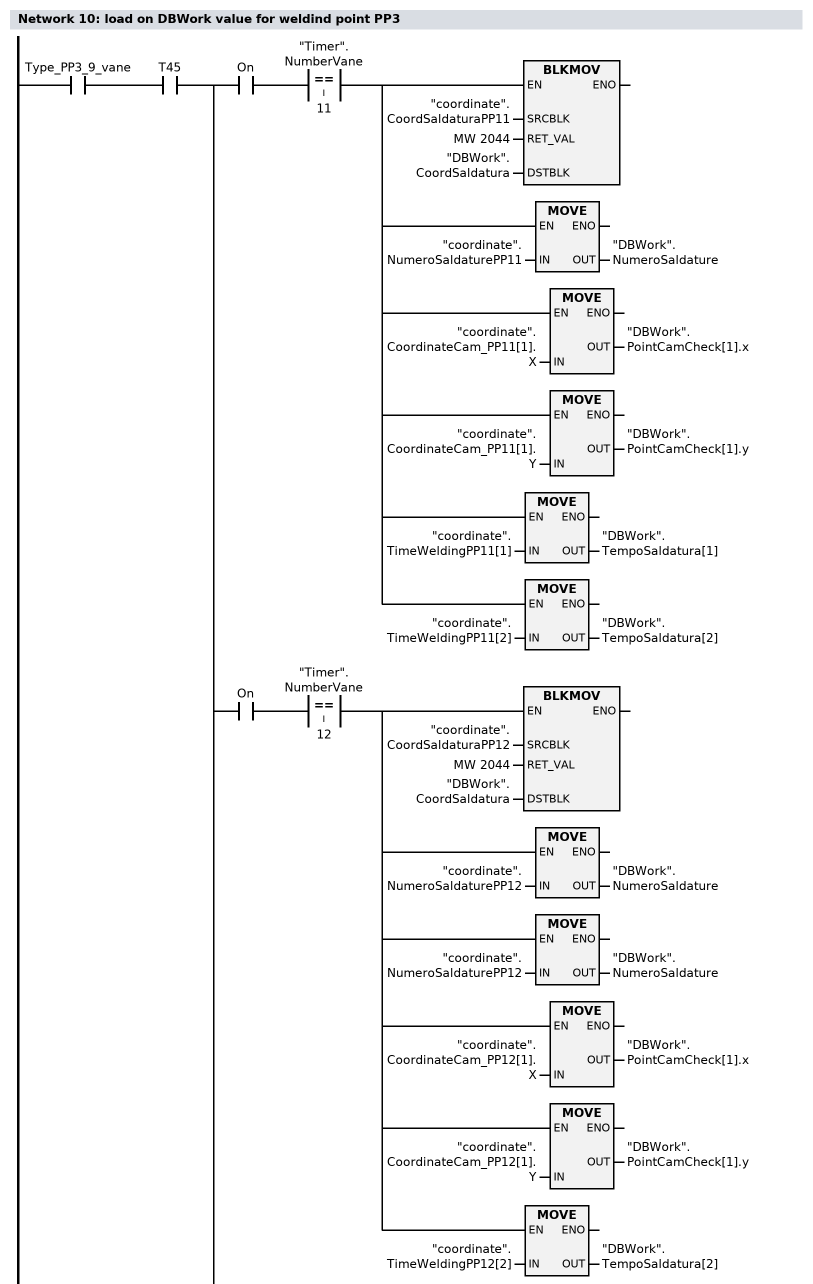
